LIN {X 0,Y 298.918,Z 266.24,A -85,B 0,C 180,E1 -16378.651,E2 -16378.651} C_VEL
LIN {X 0,Y 298.918,Z 266.244,A -85,B 0,C 180,E1 -16381.346,E2 -16381.346} C_VEL
LIN {X 0,Y 298.79,Z 266.264,A -85,B 0,C 180,E1 -16386.752,E2 -16386.752} C_VEL
LIN {X 0,Y 298.673,Z 266.281,A -85,B 0,C 180,E1 -16389.479,E2 -16389.479} C_VEL
LIN {X 0,Y 298.543,Z 266.299,A -85,B 0,C 180,E1 -16393.614,E2 -16393.614} C_VEL
LIN {X 0,Y 298.54,Z 266.293,A -85,B 0,C 180,E1 -16396.407,E2 -16396.407} C_VEL
LIN {X 0,Y 298.503,Z 266.303,A -85,B 0,C 180,E1 -16399.653,E2 -16399.653} C_VEL
LIN {X 0,Y 298.448,Z 266.307,A -85,B 0,C 180,E1 -16403.596,E2 -16403.596} C_VEL
LIN {X 0,Y 298.48,Z 266.302,A -85,B 0,C 180,E1 -16406.573,E2 -16406.573} C_VEL
LIN {X 0,Y 298.411,Z 266.31,A -85,B 0,C 180,E1 -16409.64,E2 -16409.64} C_VEL
LIN {X 0,Y 298.385,Z 266.316,A -85,B 0,C 180,E1 -16412.799,E2 -16412.799} C_VEL
LIN {X 0,Y 298.456,Z 266.307,A -85,B 0,C 180,E1 -16416.812,E2 -16416.812} C_VEL
LIN {X 0,Y 298.441,Z 266.308,A -85,B 0,C 180,E1 -16421.249,E2 -16421.249} C_VEL
LIN {X 0,Y 298.406,Z 266.315,A -85,B 0,C 180,E1 -16425.046,E2 -16425.046} C_VEL
LIN {X 0,Y 298.378,Z 266.319,A -85,B 0,C 180,E1 -16428.911,E2 -16428.911} C_VEL
LIN {X 0,Y 298.454,Z 266.306,A -85,B 0,C 180,E1 -16433.187,E2 -16433.187} C_VEL
LIN {X 0,Y 298.384,Z 266.315,A -85,B 0,C 180,E1 -16437.199,E2 -16437.199} C_VEL
LIN {X 0,Y 298.414,Z 266.315,A -85,B 0,C 180,E1 -16440.617,E2 -16440.617} C_VEL
LIN {X 0,Y 298.431,Z 266.309,A -85,B 0,C 180,E1 -16443.49,E2 -16443.49} C_VEL
LIN {X 0,Y 298.308,Z 266.328,A -85,B 0,C 180,E1 -16446.749,E2 -16446.749} C_VEL
LIN {X 0,Y 298.289,Z 266.555,A -85,B 0,C 180,E1 -16448.218,E2 -16448.218} C_VEL
LIN {X 0,Y 298.132,Z 269.038,A -85,B 0,C 180,E1 -16450.73,E2 -16450.73} C_VEL
LIN {X 0,Y 297.853,Z 273.686,A -85,B 0,C 180,E1 -16455.325,E2 -16455.325} C_VEL
LIN {X 0,Y 297.53,Z 277.67,A -85,B 0,C 180,E1 -16459.108,E2 -16459.108} C_VEL
LIN {X 0,Y 297.498,Z 279.14,A -85,B 0,C 180,E1 -16460.482,E2 -16460.482} C_VEL
LIN {X 0,Y 301.006,Z 294.207,A -85,B 0,C 180,E1 -16461.43,E2 -16461.43} C_VEL
LIN {X 0,Y 302.952,Z 305.53,A -85,B 0,C 180,E1 -16462.335,E2 -16462.335} C_VEL
LIN {X 0,Y 304.047,Z 314.476,A -85,B 0,C 180,E1 -16463.197,E2 -16463.197} C_VEL
LIN {X 0,Y 303.079,Z 325.319,A -85,B 0,C 180,E1 -16464.344,E2 -16464.344} C_VEL
LIN {X 0,Y 301.711,Z 336.458,A -85,B 0,C 180,E1 -16465.826,E2 -16465.826} C_VEL
LIN {X 0,Y 300.607,Z 345.446,A -85,B 0,C 180,E1 -16467.32,E2 -16467.32} C_VEL
LIN {X 0,Y 299.559,Z 353.696,A -85,B 0,C 180,E1 -16468.992,E2 -16468.992} C_VEL
LIN {X 0,Y 298.399,Z 361.803,A -85,B 0,C 180,E1 -16471.012,E2 -16471.012} C_VEL
LIN {X 0,Y 297.81,Z 367.29,A -85,B 0,C 180,E1 -16472.705,E2 -16472.705} C_VEL
LIN {X 0,Y 297.249,Z 372.668,A -85,B 0,C 180,E1 -16474.747,E2 -16474.747} C_VEL
LIN {X 0,Y 296.913,Z 376.869,A -85,B 0,C 180,E1 -16476.797,E2 -16476.797} C_VEL
LIN {X 0,Y 296.63,Z 379.108,A -85,B 0,C 180,E1 -16478.172,E2 -16478.172} C_VEL
LIN {X 0,Y 296.449,Z 380.852,A -85,B 0,C 180,E1 -16479.552,E2 -16479.552} C_VEL
LIN {X 0,Y 296.349,Z 382.182,A -85,B 0,C 180,E1 -16480.936,E2 -16480.936} C_VEL
LIN {X 0,Y 296.375,Z 383.581,A -85,B 0,C 180,E1 -16483.541,E2 -16483.541} C_VEL
LIN {X 0,Y 296.381,Z 383.689,A -85,B 0,C 180,E1 -16485.119,E2 -16485.119} C_VEL
LIN {X 0,Y 296.494,Z 383.364,A -85,B 0,C 180,E1 -16486.525,E2 -16486.525} C_VEL
LIN {X 0,Y 296.901,Z 381.967,A -85,B 0,C 180,E1 -16488.772,E2 -16488.772} C_VEL
LIN {X 0,Y 297.663,Z 378.824,A -85,B 0,C 180,E1 -16491.466,E2 -16491.466} C_VEL
LIN {X 0,Y 298.539,Z 375.125,A -85,B 0,C 180,E1 -16493.59,E2 -16493.59} C_VEL
LIN {X 0,Y 299.663,Z 370.217,A -85,B 0,C 180,E1 -16495.713,E2 -16495.713} C_VEL
LIN {X 0,Y 301.161,Z 363.948,A -85,B 0,C 180,E1 -16497.821,E2 -16497.821} C_VEL
LIN {X 0,Y 302.967,Z 356.064,A -85,B 0,C 180,E1 -16499.916,E2 -16499.916} C_VEL
LIN {X 0,Y 304.904,Z 347.289,A -85,B 0,C 180,E1 -16501.752,E2 -16501.752} C_VEL
LIN {X 0,Y 306.788,Z 337.818,A -85,B 0,C 180,E1 -16503.352,E2 -16503.352} C_VEL
LIN {X 0,Y 308.587,Z 327.879,A -85,B 0,C 180,E1 -16504.705,E2 -16504.705} C_VEL
LIN {X 0,Y 309.544,Z 321.191,A -85,B 0,C 180,E1 -16505.475,E2 -16505.475} C_VEL
LIN {X 0,Y 307.576,Z 309.692,A -85,B 0,C 180,E1 -16506.898,E2 -16506.898} C_VEL
LIN {X 0,Y 304.312,Z 297.366,A -85,B 0,C 180,E1 -16508.262,E2 -16508.262} C_VEL
LIN {X 0,Y 300.102,Z 285.47,A -85,B 0,C 180,E1 -16509.441,E2 -16509.441} C_VEL
LIN {X 0,Y 298.087,Z 279.79,A -85,B 0,C 180,E1 -16509.934,E2 -16509.934} C_VEL
LIN {X 0,Y 298.415,Z 276.805,A -85,B 0,C 180,E1 -16513.11,E2 -16513.11} C_VEL
LIN {X 0,Y 298.864,Z 273.306,A -85,B 0,C 180,E1 -16517.006,E2 -16517.006} C_VEL
LIN {X 0,Y 298.92,Z 271.733,A -85,B 0,C 180,E1 -16518.831,E2 -16518.831} C_VEL
LIN {X 0,Y 298.715,Z 268.955,A -85,B 0,C 180,E1 -16522.289,E2 -16522.289} C_VEL
LIN {X 0,Y 298.42,Z 266.485,A -85,B 0,C 180,E1 -16525.585,E2 -16525.585} C_VEL
LIN {X 0,Y 298.384,Z 266.322,A -85,B 0,C 180,E1 -16528.792,E2 -16528.792} C_VEL
LIN {X 0,Y 298.453,Z 266.311,A -85,B 0,C 180,E1 -16531.905,E2 -16531.905} C_VEL
LIN {X 0,Y 298.478,Z 266.304,A -85,B 0,C 180,E1 -16534.925,E2 -16534.925} C_VEL
LIN {X 0,Y 298.46,Z 266.305,A -85,B 0,C 180,E1 -16539.318,E2 -16539.318} C_VEL
LIN {X 0,Y 298.53,Z 266.295,A -85,B 0,C 180,E1 -16542.181,E2 -16542.181} C_VEL
LIN {X 0,Y 298.537,Z 266.294,A -85,B 0,C 180,E1 -16546.12,E2 -16546.12} C_VEL
LIN {X 0,Y 298.627,Z 266.288,A -85,B 0,C 180,E1 -16550.52,E2 -16550.52} C_VEL
LIN {X 0,Y 298.73,Z 266.273,A -85,B 0,C 180,E1 -16551.968,E2 -16551.968} C_VEL
LIN {X 0,Y 298.053,Z 266.359,A -85,B 0,C 180,E1 -16553.092,E2 -16553.092} C_VEL
LIN {X 0,Y 295.209,Z 266.713,A -85,B 0,C 180,E1 -16554.923,E2 -16554.923} C_VEL
LIN {X 0,Y 292.837,Z 267.009,A -85,B 0,C 180,E1 -16556.409,E2 -16556.409} C_VEL
LIN {X 0,Y 291.867,Z 267.129,A -85,B 0,C 180,E1 -16557.56,E2 -16557.56} C_VEL
LIN {X 0,Y 291.812,Z 267.134,A -85,B 0,C 180,E1 -16557.949,E2 -16557.949} C_VEL
LIN {X 0,Y 291.944,Z 267.118,A -85,B 0,C 180,E1 -16560.002,E2 -16560.002} C_VEL
LIN {X 0,Y 291.783,Z 267.14,A -85,B 0,C 180,E1 -16562.763,E2 -16562.763} C_VEL
LIN {X 0,Y 291.739,Z 267.146,A -85,B 0,C 180,E1 -16566.92,E2 -16566.92} C_VEL
LIN {X 0,Y 291.624,Z 267.159,A -85,B 0,C 180,E1 -16569.714,E2 -16569.714} C_VEL
LIN {X 0,Y 291.517,Z 267.174,A -85,B 0,C 180,E1 -16573.952,E2 -16573.952} C_VEL
LIN {X 0,Y 291.483,Z 267.181,A -85,B 0,C 180,E1 -16576.82,E2 -16576.82} C_VEL
LIN {X 0,Y 291.448,Z 267.187,A -85,B 0,C 180,E1 -16579.877,E2 -16579.877} C_VEL
LIN {X 0,Y 291.369,Z 267.197,A -85,B 0,C 180,E1 -16584.21,E2 -16584.21} C_VEL
LIN {X 0,Y 291.393,Z 267.195,A -85,B 0,C 180,E1 -16587.276,E2 -16587.276} C_VEL
LIN {X 0,Y 291.319,Z 267.202,A -85,B 0,C 180,E1 -16590.44,E2 -16590.44} C_VEL
LIN {X 0,Y 291.342,Z 267.196,A -85,B 0,C 180,E1 -16593.7,E2 -16593.7} C_VEL
LIN {X 0,Y 291.375,Z 267.191,A -85,B 0,C 180,E1 -16597.255,E2 -16597.255} C_VEL
LIN {X 0,Y 291.379,Z 267.265,A -85,B 0,C 180,E1 -16598.411,E2 -16598.411} C_VEL
LIN {X 0,Y 291.89,Z 270.67,A -85,B 0,C 180,E1 -16602.392,E2 -16602.392} C_VEL
LIN {X 0,Y 292.517,Z 274.169,A -85,B 0,C 180,E1 -16606.121,E2 -16606.121} C_VEL
LIN {X 0,Y 293.083,Z 277.742,A -85,B 0,C 180,E1 -16609.652,E2 -16609.652} C_VEL
LIN {X 0,Y 293.435,Z 281.675,A -85,B 0,C 180,E1 -16613.219,E2 -16613.219} C_VEL
LIN {X 0,Y 293.336,Z 283.651,A -85,B 0,C 180,E1 -16614.901,E2 -16614.901} C_VEL
LIN {X 0,Y 292.655,Z 287.637,A -85,B 0,C 180,E1 -16618.109,E2 -16618.109} C_VEL
LIN {X 0,Y 291.73,Z 293.108,A -85,B 0,C 180,E1 -16622.337,E2 -16622.337} C_VEL
LIN {X 0,Y 292.705,Z 296.464,A -85,B 0,C 180,E1 -16622.601,E2 -16622.601} C_VEL
LIN {X 0,Y 296.744,Z 309.875,A -85,B 0,C 180,E1 -16623.81,E2 -16623.81} C_VEL
LIN {X 0,Y 299.461,Z 322.339,A -85,B 0,C 180,E1 -16625.088,E2 -16625.088} C_VEL
LIN {X 0,Y 301.014,Z 333.959,A -85,B 0,C 180,E1 -16626.455,E2 -16626.455} C_VEL
LIN {X 0,Y 301.385,Z 342.41,A -85,B 0,C 180,E1 -16627.552,E2 -16627.552} C_VEL
LIN {X 0,Y 299.351,Z 353.181,A -85,B 0,C 180,E1 -16629.021,E2 -16629.021} C_VEL
LIN {X 0,Y 297.151,Z 362.889,A -85,B 0,C 180,E1 -16630.664,E2 -16630.664} C_VEL
LIN {X 0,Y 295.31,Z 371.442,A -85,B 0,C 180,E1 -16632.477,E2 -16632.477} C_VEL
LIN {X 0,Y 293.712,Z 378.715,A -85,B 0,C 180,E1 -16634.384,E2 -16634.384} C_VEL
LIN {X 0,Y 292.344,Z 384.053,A -85,B 0,C 180,E1 -16636.09,E2 -16636.09} C_VEL
LIN {X 0,Y 291.181,Z 389.297,A -85,B 0,C 180,E1 -16638.162,E2 -16638.162} C_VEL
LIN {X 0,Y 290.347,Z 393.396,A -85,B 0,C 180,E1 -16640.245,E2 -16640.245} C_VEL
LIN {X 0,Y 289.935,Z 395.563,A -85,B 0,C 180,E1 -16641.638,E2 -16641.638} C_VEL
LIN {X 0,Y 289.482,Z 398.581,A -85,B 0,C 180,E1 -16644.427,E2 -16644.427} C_VEL
LIN {X 0,Y 289.406,Z 399.505,A -85,B 0,C 180,E1 -16645.822,E2 -16645.822} C_VEL
LIN {X 0,Y 289.433,Z 400.027,A -85,B 0,C 180,E1 -16647.217,E2 -16647.217} C_VEL
LIN {X 0,Y 289.409,Z 400.124,A -85,B 0,C 180,E1 -16648.609,E2 -16648.609} C_VEL
LIN {X 0,Y 289.439,Z 399.839,A -85,B 0,C 180,E1 -16650,E2 -16650} C_VEL
LIN {X 0,Y 289.423,Z 399.164,A -85,B 0,C 180,E1 -16651.391,E2 -16651.391} C_VEL
LIN {X 0,Y 289.47,Z 398.086,A -85,B 0,C 180,E1 -16652.783,E2 -16652.783} C_VEL
LIN {X 0,Y 289.445,Z 396.547,A -85,B 0,C 180,E1 -16654.177,E2 -16654.177} C_VEL
LIN {X 0,Y 289.564,Z 393.444,A -85,B 0,C 180,E1 -16656.27,E2 -16656.27} C_VEL
LIN {X 0,Y 289.839,Z 389.262,A -85,B 0,C 180,E1 -16658.365,E2 -16658.365} C_VEL
LIN {X 0,Y 290.461,Z 382.866,A -85,B 0,C 180,E1 -16660.808,E2 -16660.808} C_VEL
LIN {X 0,Y 291.276,Z 375.883,A -85,B 0,C 180,E1 -16662.896,E2 -16662.896} C_VEL
LIN {X 0,Y 292.21,Z 368.739,A -85,B 0,C 180,E1 -16664.627,E2 -16664.627} C_VEL
LIN {X 0,Y 293.307,Z 359.865,A -85,B 0,C 180,E1 -16666.39,E2 -16666.39} C_VEL
LIN {X 0,Y 294.579,Z 349.371,A -85,B 0,C 180,E1 -16668.068,E2 -16668.068} C_VEL
LIN {X 0,Y 295.97,Z 338.769,A -85,B 0,C 180,E1 -16669.416,E2 -16669.416} C_VEL
LIN {X 0,Y 295.933,Z 333.974,A -85,B 0,C 180,E1 -16669.961,E2 -16669.961} C_VEL
LIN {X 0,Y 294.798,Z 321.713,A -85,B 0,C 180,E1 -16671.185,E2 -16671.185} C_VEL
LIN {X 0,Y 293.106,Z 308.712,A -85,B 0,C 180,E1 -16672.196,E2 -16672.196} C_VEL
LIN {X 0,Y 290.789,Z 295.542,A -85,B 0,C 180,E1 -16672.971,E2 -16672.971} C_VEL
LIN {X 0,Y 290.508,Z 293.683,A -85,B 0,C 180,E1 -16673.097,E2 -16673.097} C_VEL
LIN {X 0,Y 291.1,Z 287.723,A -85,B 0,C 180,E1 -16677.304,E2 -16677.304} C_VEL
LIN {X 0,Y 291.952,Z 281.246,A -85,B 0,C 180,E1 -16681.977,E2 -16681.977} C_VEL
LIN {X 0,Y 292.563,Z 276.873,A -85,B 0,C 180,E1 -16685.237,E2 -16685.237} C_VEL
LIN {X 0,Y 292.569,Z 273.875,A -85,B 0,C 180,E1 -16687.558,E2 -16687.558} C_VEL
LIN {X 0,Y 291.704,Z 268.923,A -85,B 0,C 180,E1 -16691.677,E2 -16691.677} C_VEL
LIN {X 0,Y 291.356,Z 267.194,A -85,B 0,C 180,E1 -16693.335,E2 -16693.335} C_VEL
LIN {X 0,Y 291.283,Z 267.203,A -85,B 0,C 180,E1 -16697.499,E2 -16697.499} C_VEL
LIN {X 0,Y 291.331,Z 267.197,A -85,B 0,C 180,E1 -16701.153,E2 -16701.153} C_VEL
LIN {X 0,Y 291.353,Z 267.195,A -85,B 0,C 180,E1 -16704.623,E2 -16704.623} C_VEL
LIN {X 0,Y 291.364,Z 267.189,A -85,B 0,C 180,E1 -16707.948,E2 -16707.948} C_VEL
LIN {X 0,Y 291.341,Z 267.192,A -85,B 0,C 180,E1 -16711.152,E2 -16711.152} C_VEL
LIN {X 0,Y 291.356,Z 267.193,A -85,B 0,C 180,E1 -16714.265,E2 -16714.265} C_VEL
LIN {X 0,Y 291.363,Z 267.189,A -85,B 0,C 180,E1 -16717.296,E2 -16717.296} C_VEL
LIN {X 0,Y 291.455,Z 267.182,A -85,B 0,C 180,E1 -16720.268,E2 -16720.268} C_VEL
LIN {X 0,Y 291.537,Z 267.17,A -85,B 0,C 180,E1 -16724.633,E2 -16724.633} C_VEL
LIN {X 0,Y 291.53,Z 267.167,A -85,B 0,C 180,E1 -16728.879,E2 -16728.879} C_VEL
LIN {X 0,Y 291.683,Z 267.151,A -85,B 0,C 180,E1 -16731.686,E2 -16731.686} C_VEL
LIN {X 0,Y 291.621,Z 267.157,A -85,B 0,C 180,E1 -16734.467,E2 -16734.467} C_VEL
LIN {X 0,Y 291.884,Z 267.115,A -85,B 0,C 180,E1 -16738.619,E2 -16738.619} C_VEL
LIN {X 0,Y 291.885,Z 267.119,A -85,B 0,C 180,E1 -16741.378,E2 -16741.378} C_VEL
LIN {X 0,Y 291.739,Z 267.142,A -85,B 0,C 180,E1 -16746.916,E2 -16746.916} C_VEL
LIN {X 0,Y 291.622,Z 267.159,A -85,B 0,C 180,E1 -16749.71,E2 -16749.71} C_VEL
LIN {X 0,Y 291.513,Z 267.172,A -85,B 0,C 180,E1 -16753.949,E2 -16753.949} C_VEL
LIN {X 0,Y 291.478,Z 267.173,A -85,B 0,C 180,E1 -16756.816,E2 -16756.816} C_VEL
LIN {X 0,Y 291.442,Z 267.181,A -85,B 0,C 180,E1 -16759.873,E2 -16759.873} C_VEL
LIN {X 0,Y 291.391,Z 267.183,A -85,B 0,C 180,E1 -16764.204,E2 -16764.204} C_VEL
LIN {X 0,Y 291.413,Z 267.187,A -85,B 0,C 180,E1 -16767.27,E2 -16767.27} C_VEL
LIN {X 0,Y 291.328,Z 267.191,A -85,B 0,C 180,E1 -16770.436,E2 -16770.436} C_VEL
LIN {X 0,Y 291.335,Z 267.193,A -85,B 0,C 180,E1 -16773.697,E2 -16773.697} C_VEL
LIN {X 0,Y 291.389,Z 267.188,A -85,B 0,C 180,E1 -16777.259,E2 -16777.259} C_VEL
LIN {X 0,Y 291.39,Z 267.188,A -85,B 0,C 180,E1 -16780.63,E2 -16780.63} C_VEL
LIN {X 0,Y 291.342,Z 267.192,A -85,B 0,C 180,E1 -16784.389,E2 -16784.389} C_VEL
LIN {X 0,Y 291.321,Z 267.194,A -85,B 0,C 180,E1 -16788.402,E2 -16788.402} C_VEL
LIN {X 0,Y 291.343,Z 267.192,A -85,B 0,C 180,E1 -16791.158,E2 -16791.158} C_VEL
LIN {X 0,Y 291.375,Z 267.193,A -85,B 0,C 180,E1 -16794.629,E2 -16794.629} C_VEL
LIN {X 0,Y 291.359,Z 267.191,A -85,B 0,C 180,E1 -16797.95,E2 -16797.95} C_VEL
LIN {X 0,Y 291.358,Z 267.19,A -85,B 0,C 180,E1 -16801.156,E2 -16801.156} C_VEL
LIN {X 0,Y 291.354,Z 267.194,A -85,B 0,C 180,E1 -16804.267,E2 -16804.267} C_VEL
LIN {X 0,Y 291.293,Z 267.305,A -85,B 0,C 180,E1 -16808.04,E2 -16808.04} C_VEL
LIN {X 0,Y 290.956,Z 270.87,A -85,B 0,C 180,E1 -16811.699,E2 -16811.699} C_VEL
LIN {X 0,Y 290.72,Z 275.198,A -85,B 0,C 180,E1 -16816.011,E2 -16816.011} C_VEL
LIN {X 0,Y 290.437,Z 279.352,A -85,B 0,C 180,E1 -16820.028,E2 -16820.028} C_VEL
LIN {X 0,Y 293.921,Z 293.917,A -85,B 0,C 180,E1 -16820.969,E2 -16820.969} C_VEL
LIN {X 0,Y 296.064,Z 306.265,A -85,B 0,C 180,E1 -16821.983,E2 -16821.983} C_VEL
LIN {X 0,Y 297.199,Z 316.77,A -85,B 0,C 180,E1 -16823.039,E2 -16823.039} C_VEL
LIN {X 0,Y 295.841,Z 328.512,A -85,B 0,C 180,E1 -16824.376,E2 -16824.376} C_VEL
LIN {X 0,Y 294.493,Z 339.037,A -85,B 0,C 180,E1 -16825.894,E2 -16825.894} C_VEL
LIN {X 0,Y 293.248,Z 348.521,A -85,B 0,C 180,E1 -16827.596,E2 -16827.596} C_VEL
LIN {X 0,Y 292.035,Z 357.643,A -85,B 0,C 180,E1 -16829.655,E2 -16829.655} C_VEL
LIN {X 0,Y 291.013,Z 365.006,A -85,B 0,C 180,E1 -16831.73,E2 -16831.73} C_VEL
LIN {X 0,Y 290.457,Z 369.991,A -85,B 0,C 180,E1 -16833.468,E2 -16833.468} C_VEL
LIN {X 0,Y 290.011,Z 374.834,A -85,B 0,C 180,E1 -16835.562,E2 -16835.562} C_VEL
LIN {X 0,Y 289.641,Z 378.568,A -85,B 0,C 180,E1 -16837.669,E2 -16837.669} C_VEL
LIN {X 0,Y 289.332,Z 381.283,A -85,B 0,C 180,E1 -16839.789,E2 -16839.789} C_VEL
LIN {X 0,Y 289.265,Z 382.561,A -85,B 0,C 180,E1 -16841.207,E2 -16841.207} C_VEL
LIN {X 0,Y 289.284,Z 383.782,A -85,B 0,C 180,E1 -16843.654,E2 -16843.654} C_VEL
LIN {X 0,Y 289.308,Z 383.868,A -85,B 0,C 180,E1 -16845.498,E2 -16845.498} C_VEL
LIN {X 0,Y 289.457,Z 383.493,A -85,B 0,C 180,E1 -16846.939,E2 -16846.939} C_VEL
LIN {X 0,Y 289.857,Z 382.191,A -85,B 0,C 180,E1 -16848.991,E2 -16848.991} C_VEL
LIN {X 0,Y 290.756,Z 378.689,A -85,B 0,C 180,E1 -16852.003,E2 -16852.003} C_VEL
LIN {X 0,Y 291.745,Z 374.873,A -85,B 0,C 180,E1 -16854.174,E2 -16854.174} C_VEL
LIN {X 0,Y 292.983,Z 369.841,A -85,B 0,C 180,E1 -16856.344,E2 -16856.344} C_VEL
LIN {X 0,Y 294.605,Z 363.436,A -85,B 0,C 180,E1 -16858.496,E2 -16858.496} C_VEL
LIN {X 0,Y 296.177,Z 356.815,A -85,B 0,C 180,E1 -16860.28,E2 -16860.28} C_VEL
LIN {X 0,Y 298.24,Z 347.959,A -85,B 0,C 180,E1 -16862.199,E2 -16862.199} C_VEL
LIN {X 0,Y 300.393,Z 337.762,A -85,B 0,C 180,E1 -16863.957,E2 -16863.957} C_VEL
LIN {X 0,Y 302.262,Z 327.768,A -85,B 0,C 180,E1 -16865.335,E2 -16865.335} C_VEL
LIN {X 0,Y 302.962,Z 323.772,A -85,B 0,C 180,E1 -16865.802,E2 -16865.802} C_VEL
LIN {X 0,Y 302.229,Z 317.404,A -85,B 0,C 180,E1 -16866.658,E2 -16866.658} C_VEL
LIN {X 0,Y 300.306,Z 307.817,A -85,B 0,C 180,E1 -16867.854,E2 -16867.854} C_VEL
LIN {X 0,Y 297.266,Z 296.818,A -85,B 0,C 180,E1 -16869.098,E2 -16869.098} C_VEL
LIN {X 0,Y 292.499,Z 283.66,A -85,B 0,C 180,E1 -16870.43,E2 -16870.43} C_VEL
LIN {X 0,Y 291.299,Z 280.869,A -85,B 0,C 180,E1 -16870.707,E2 -16870.707} C_VEL
LIN {X 0,Y 291.157,Z 279.995,A -85,B 0,C 180,E1 -16870.796,E2 -16870.796} C_VEL
LIN {X 0,Y 291.511,Z 276.756,A -85,B 0,C 180,E1 -16874.358,E2 -16874.358} C_VEL
LIN {X 0,Y 291.862,Z 273.931,A -85,B 0,C 180,E1 -16877.608,E2 -16877.608} C_VEL
LIN {X 0,Y 291.817,Z 271.01,A -85,B 0,C 180,E1 -16881.234,E2 -16881.234} C_VEL
LIN {X 0,Y 291.497,Z 268.156,A -85,B 0,C 180,E1 -16885.057,E2 -16885.057} C_VEL
LIN {X 0,Y 291.346,Z 267.287,A -85,B 0,C 180,E1 -16886.304,E2 -16886.304} C_VEL
LIN {X 0,Y 291.377,Z 267.193,A -85,B 0,C 180,E1 -16890.261,E2 -16890.261} C_VEL
LIN {X 0,Y 291.409,Z 267.187,A -85,B 0,C 180,E1 -16894.273,E2 -16894.273} C_VEL
LIN {X 0,Y 291.39,Z 267.185,A -85,B 0,C 180,E1 -16897.302,E2 -16897.302} C_VEL
LIN {X 0,Y 291.495,Z 267.174,A -85,B 0,C 180,E1 -16900.275,E2 -16900.275} C_VEL
LIN {X 0,Y 291.532,Z 267.17,A -85,B 0,C 180,E1 -16904.636,E2 -16904.636} C_VEL
LIN {X 0,Y 291.527,Z 267.172,A -85,B 0,C 180,E1 -16908.882,E2 -16908.882} C_VEL
LIN {X 0,Y 291.675,Z 267.151,A -85,B 0,C 180,E1 -16911.967,E2 -16911.967} C_VEL
LIN {X 0,Y 291.619,Z 267.161,A -85,B 0,C 180,E1 -16914.47,E2 -16914.47} C_VEL
LIN {X 0,Y 291.812,Z 267.134,A -85,B 0,C 180,E1 -16917.949,E2 -16917.949} C_VEL
LIN {X 0,Y 291.205,Z 267.212,A -85,B 0,C 180,E1 -16919.102,E2 -16919.102} C_VEL
LIN {X 0,Y 288.33,Z 267.57,A -85,B 0,C 180,E1 -16920.977,E2 -16920.977} C_VEL
LIN {X 0,Y 285.802,Z 267.885,A -85,B 0,C 180,E1 -16922.499,E2 -16922.499} C_VEL
LIN {X 0,Y 284.649,Z 268.028,A -85,B 0,C 180,E1 -16923.679,E2 -16923.679} C_VEL
LIN {X 0,Y 284.521,Z 268.043,A -85,B 0,C 180,E1 -16924.081,E2 -16924.081} C_VEL
LIN {X 0,Y 284.692,Z 268.023,A -85,B 0,C 180,E1 -16927.092,E2 -16927.092} C_VEL
LIN {X 0,Y 284.561,Z 268.039,A -85,B 0,C 180,E1 -16929.957,E2 -16929.957} C_VEL
LIN {X 0,Y 284.473,Z 268.054,A -85,B 0,C 180,E1 -16934.305,E2 -16934.305} C_VEL
LIN {X 0,Y 284.421,Z 268.06,A -85,B 0,C 180,E1 -16937.25,E2 -16937.25} C_VEL
LIN {X 0,Y 284.376,Z 268.068,A -85,B 0,C 180,E1 -16940.244,E2 -16940.244} C_VEL
LIN {X 0,Y 284.319,Z 268.076,A -85,B 0,C 180,E1 -16944.85,E2 -16944.85} C_VEL
LIN {X 0,Y 284.304,Z 268.077,A -85,B 0,C 180,E1 -16948.015,E2 -16948.015} C_VEL
LIN {X 0,Y 284.284,Z 268.078,A -85,B 0,C 180,E1 -16951.277,E2 -16951.277} C_VEL
LIN {X 0,Y 284.34,Z 268.067,A -85,B 0,C 180,E1 -16955.35,E2 -16955.35} C_VEL
LIN {X 0,Y 284.359,Z 268.264,A -85,B 0,C 180,E1 -16957.733,E2 -16957.733} C_VEL
LIN {X 0,Y 284.689,Z 270.141,A -85,B 0,C 180,E1 -16960.069,E2 -16960.069} C_VEL
LIN {X 0,Y 285.256,Z 273.914,A -85,B 0,C 180,E1 -16964.4,E2 -16964.4} C_VEL
LIN {X 0,Y 285.922,Z 277.77,A -85,B 0,C 180,E1 -16968.421,E2 -16968.421} C_VEL
LIN {X 0,Y 286.427,Z 281.698,A -85,B 0,C 180,E1 -16972.164,E2 -16972.164} C_VEL
LIN {X 0,Y 286.373,Z 283.86,A -85,B 0,C 180,E1 -16974.085,E2 -16974.085} C_VEL
LIN {X 0,Y 285.837,Z 287.621,A -85,B 0,C 180,E1 -16977.254,E2 -16977.254} C_VEL
LIN {X 0,Y 284.839,Z 292.896,A -85,B 0,C 180,E1 -16981.465,E2 -16981.465} C_VEL
LIN {X 0,Y 285.781,Z 296.152,A -85,B 0,C 180,E1 -16981.723,E2 -16981.723} C_VEL
LIN {X 0,Y 289.823,Z 309.168,A -85,B 0,C 180,E1 -16982.962,E2 -16982.962} C_VEL
LIN {X 0,Y 292.471,Z 320.562,A -85,B 0,C 180,E1 -16984.174,E2 -16984.174} C_VEL
LIN {X 0,Y 294.185,Z 332.406,A -85,B 0,C 180,E1 -16985.581,E2 -16985.581} C_VEL
LIN {X 0,Y 294.795,Z 341.735,A -85,B 0,C 180,E1 -16986.837,E2 -16986.837} C_VEL
LIN {X 0,Y 294.451,Z 345.58,A -85,B 0,C 180,E1 -16987.365,E2 -16987.365} C_VEL
LIN {X 0,Y 292.241,Z 355.763,A -85,B 0,C 180,E1 -16988.856,E2 -16988.856} C_VEL
LIN {X 0,Y 290.058,Z 364.936,A -85,B 0,C 180,E1 -16990.54,E2 -16990.54} C_VEL
LIN {X 0,Y 288.311,Z 372.947,A -85,B 0,C 180,E1 -16992.378,E2 -16992.378} C_VEL
LIN {X 0,Y 286.582,Z 379.973,A -85,B 0,C 180,E1 -16994.351,E2 -16994.351} C_VEL
LIN {X 0,Y 284.968,Z 385.995,A -85,B 0,C 180,E1 -16996.45,E2 -16996.45} C_VEL
LIN {X 0,Y 283.873,Z 390.783,A -85,B 0,C 180,E1 -16998.577,E2 -16998.577} C_VEL
LIN {X 0,Y 283.102,Z 394.477,A -85,B 0,C 180,E1 -17000.714,E2 -17000.714} C_VEL
LIN {X 0,Y 282.588,Z 397.178,A -85,B 0,C 180,E1 -17002.857,E2 -17002.857} C_VEL
LIN {X 0,Y 282.401,Z 398.677,A -85,B 0,C 180,E1 -17004.553,E2 -17004.553} C_VEL
LIN {X 0,Y 282.339,Z 399.838,A -85,B 0,C 180,E1 -17007.147,E2 -17007.147} C_VEL
LIN {X 0,Y 282.333,Z 399.912,A -85,B 0,C 180,E1 -17008.574,E2 -17008.574} C_VEL
LIN {X 0,Y 282.358,Z 399.602,A -85,B 0,C 180,E1 -17010,E2 -17010} C_VEL
LIN {X 0,Y 282.346,Z 398.904,A -85,B 0,C 180,E1 -17011.426,E2 -17011.426} C_VEL
LIN {X 0,Y 282.375,Z 397.778,A -85,B 0,C 180,E1 -17012.853,E2 -17012.853} C_VEL
LIN {X 0,Y 282.413,Z 394.583,A -85,B 0,C 180,E1 -17015.474,E2 -17015.474} C_VEL
LIN {X 0,Y 282.673,Z 390.358,A -85,B 0,C 180,E1 -17017.859,E2 -17017.859} C_VEL
LIN {X 0,Y 283.127,Z 385.342,A -85,B 0,C 180,E1 -17020.006,E2 -17020.006} C_VEL
LIN {X 0,Y 283.796,Z 379.02,A -85,B 0,C 180,E1 -17022.151,E2 -17022.151} C_VEL
LIN {X 0,Y 284.94,Z 371.097,A -85,B 0,C 180,E1 -17024.279,E2 -17024.279} C_VEL
LIN {X 0,Y 286.143,Z 361.996,A -85,B 0,C 180,E1 -17026.242,E2 -17026.242} C_VEL
LIN {X 0,Y 287.369,Z 351.995,A -85,B 0,C 180,E1 -17027.984,E2 -17027.984} C_VEL
LIN {X 0,Y 288.671,Z 342.007,A -85,B 0,C 180,E1 -17029.372,E2 -17029.372} C_VEL
LIN {X 0,Y 289.22,Z 337.68,A -85,B 0,C 180,E1 -17029.888,E2 -17029.888} C_VEL
LIN {X 0,Y 288.286,Z 325.951,A -85,B 0,C 180,E1 -17031.182,E2 -17031.182} C_VEL
LIN {X 0,Y 286.91,Z 313.75,A -85,B 0,C 180,E1 -17032.258,E2 -17032.258} C_VEL
LIN {X 0,Y 284.839,Z 300.778,A -85,B 0,C 180,E1 -17033.149,E2 -17033.149} C_VEL
LIN {X 0,Y 283.475,Z 293.526,A -85,B 0,C 180,E1 -17033.544,E2 -17033.544} C_VEL
LIN {X 0,Y 284.116,Z 287.357,A -85,B 0,C 180,E1 -17038.033,E2 -17038.033} C_VEL
LIN {X 0,Y 284.915,Z 281.979,A -85,B 0,C 180,E1 -17042.028,E2 -17042.028} C_VEL
LIN {X 0,Y 285.555,Z 277.196,A -85,B 0,C 180,E1 -17045.688,E2 -17045.688} C_VEL
LIN {X 0,Y 285.449,Z 274.292,A -85,B 0,C 180,E1 -17048.011,E2 -17048.011} C_VEL
LIN {X 0,Y 284.615,Z 269.424,A -85,B 0,C 180,E1 -17052.199,E2 -17052.199} C_VEL
LIN {X 0,Y 284.317,Z 268.071,A -85,B 0,C 180,E1 -17053.487,E2 -17053.487} C_VEL
LIN {X 0,Y 284.233,Z 268.081,A -85,B 0,C 180,E1 -17058.116,E2 -17058.116} C_VEL
LIN {X 0,Y 284.292,Z 268.072,A -85,B 0,C 180,E1 -17061.826,E2 -17061.826} C_VEL
LIN {X 0,Y 284.305,Z 268.069,A -85,B 0,C 180,E1 -17065.349,E2 -17065.349} C_VEL
LIN {X 0,Y 284.283,Z 268.074,A -85,B 0,C 180,E1 -17068.723,E2 -17068.723} C_VEL
LIN {X 0,Y 284.281,Z 268.072,A -85,B 0,C 180,E1 -17071.982,E2 -17071.982} C_VEL
LIN {X 0,Y 284.318,Z 268.068,A -85,B 0,C 180,E1 -17076.145,E2 -17076.145} C_VEL
LIN {X 0,Y 284.385,Z 268.06,A -85,B 0,C 180,E1 -17079.896,E2 -17079.896} C_VEL
LIN {X 0,Y 284.475,Z 268.051,A -85,B 0,C 180,E1 -17084.468,E2 -17084.468} C_VEL
LIN {X 0,Y 284.482,Z 268.046,A -85,B 0,C 180,E1 -17088.6,E2 -17088.6} C_VEL
LIN {X 0,Y 284.634,Z 268.028,A -85,B 0,C 180,E1 -17091.479,E2 -17091.479} C_VEL
LIN {X 0,Y 284.591,Z 268.034,A -85,B 0,C 180,E1 -17094.329,E2 -17094.329} C_VEL
LIN {X 0,Y 284.85,Z 267.99,A -85,B 0,C 180,E1 -17098.585,E2 -17098.585} C_VEL
LIN {X 0,Y 284.85,Z 267.995,A -85,B 0,C 180,E1 -17101.412,E2 -17101.412} C_VEL
LIN {X 0,Y 284.691,Z 268.021,A -85,B 0,C 180,E1 -17107.088,E2 -17107.088} C_VEL
LIN {X 0,Y 284.559,Z 268.037,A -85,B 0,C 180,E1 -17109.954,E2 -17109.954} C_VEL
LIN {X 0,Y 284.47,Z 268.048,A -85,B 0,C 180,E1 -17114.301,E2 -17114.301} C_VEL
LIN {X 0,Y 284.417,Z 268.055,A -85,B 0,C 180,E1 -17117.247,E2 -17117.247} C_VEL
LIN {X 0,Y 284.37,Z 268.06,A -85,B 0,C 180,E1 -17120.241,E2 -17120.241} C_VEL
LIN {X 0,Y 284.36,Z 268.06,A -85,B 0,C 180,E1 -17123.874,E2 -17123.874} C_VEL
LIN {X 0,Y 284.388,Z 268.062,A -85,B 0,C 180,E1 -17127.172,E2 -17127.172} C_VEL
LIN {X 0,Y 284.286,Z 268.073,A -85,B 0,C 180,E1 -17131.273,E2 -17131.273} C_VEL
LIN {X 0,Y 284.352,Z 268.063,A -85,B 0,C 180,E1 -17135.353,E2 -17135.353} C_VEL
LIN {X 0,Y 284.321,Z 268.065,A -85,B 0,C 180,E1 -17138.165,E2 -17138.165} C_VEL
LIN {X 0,Y 284.33,Z 268.063,A -85,B 0,C 180,E1 -17142.139,E2 -17142.139} C_VEL
LIN {X 0,Y 284.286,Z 268.071,A -85,B 0,C 180,E1 -17146.196,E2 -17146.196} C_VEL
LIN {X 0,Y 284.296,Z 268.07,A -85,B 0,C 180,E1 -17150.023,E2 -17150.023} C_VEL
LIN {X 0,Y 284.337,Z 268.064,A -85,B 0,C 180,E1 -17153.616,E2 -17153.616} C_VEL
LIN {X 0,Y 284.297,Z 268.07,A -85,B 0,C 180,E1 -17157.189,E2 -17157.189} C_VEL
LIN {X 0,Y 284.343,Z 268.068,A -85,B 0,C 180,E1 -17160.375,E2 -17160.375} C_VEL
LIN {X 0,Y 284.335,Z 268.065,A -85,B 0,C 180,E1 -17163.583,E2 -17163.583} C_VEL
LIN {X 0,Y 284.265,Z 268.232,A -85,B 0,C 180,E1 -17168.042,E2 -17168.042} C_VEL
LIN {X 0,Y 283.953,Z 271.263,A -85,B 0,C 180,E1 -17171.231,E2 -17171.231} C_VEL
LIN {X 0,Y 283.682,Z 275.615,A -85,B 0,C 180,E1 -17175.656,E2 -17175.656} C_VEL
LIN {X 0,Y 283.383,Z 279.567,A -85,B 0,C 180,E1 -17179.554,E2 -17179.554} C_VEL
LIN {X 0,Y 286.792,Z 293.525,A -85,B 0,C 180,E1 -17180.475,E2 -17180.475} C_VEL
LIN {X 0,Y 289.007,Z 305.951,A -85,B 0,C 180,E1 -17181.519,E2 -17181.519} C_VEL
LIN {X 0,Y 290.253,Z 315.704,A -85,B 0,C 180,E1 -17182.522,E2 -17182.522} C_VEL
LIN {X 0,Y 289.816,Z 322.077,A -85,B 0,C 180,E1 -17183.211,E2 -17183.211} C_VEL
LIN {X 0,Y 288.461,Z 332.762,A -85,B 0,C 180,E1 -17184.583,E2 -17184.583} C_VEL
LIN {X 0,Y 287.249,Z 342.478,A -85,B 0,C 180,E1 -17186.142,E2 -17186.142} C_VEL
LIN {X 0,Y 285.9,Z 351.363,A -85,B 0,C 180,E1 -17187.887,E2 -17187.887} C_VEL
LIN {X 0,Y 284.886,Z 358.679,A -85,B 0,C 180,E1 -17189.647,E2 -17189.647} C_VEL
LIN {X 0,Y 283.92,Z 365.887,A -85,B 0,C 180,E1 -17191.773,E2 -17191.773} C_VEL
LIN {X 0,Y 283.319,Z 370.75,A -85,B 0,C 180,E1 -17193.555,E2 -17193.555} C_VEL
LIN {X 0,Y 282.893,Z 375.474,A -85,B 0,C 180,E1 -17195.703,E2 -17195.703} C_VEL
LIN {X 0,Y 282.496,Z 379.102,A -85,B 0,C 180,E1 -17197.864,E2 -17197.864} C_VEL
LIN {X 0,Y 282.209,Z 381.712,A -85,B 0,C 180,E1 -17200.039,E2 -17200.039} C_VEL
LIN {X 0,Y 282.161,Z 382.935,A -85,B 0,C 180,E1 -17201.493,E2 -17201.493} C_VEL
LIN {X 0,Y 282.194,Z 383.982,A -85,B 0,C 180,E1 -17203.773,E2 -17203.773} C_VEL
LIN {X 0,Y 282.236,Z 384.047,A -85,B 0,C 180,E1 -17205.897,E2 -17205.897} C_VEL
LIN {X 0,Y 282.45,Z 383.6,A -85,B 0,C 180,E1 -17207.372,E2 -17207.372} C_VEL
LIN {X 0,Y 282.817,Z 382.415,A -85,B 0,C 180,E1 -17209.22,E2 -17209.22} C_VEL
LIN {X 0,Y 283.595,Z 379.637,A -85,B 0,C 180,E1 -17211.822,E2 -17211.822} C_VEL
LIN {X 0,Y 284.516,Z 376.266,A -85,B 0,C 180,E1 -17213.947,E2 -17213.947} C_VEL
LIN {X 0,Y 285.83,Z 371.334,A -85,B 0,C 180,E1 -17216.268,E2 -17216.268} C_VEL
LIN {X 0,Y 287.618,Z 364.65,A -85,B 0,C 180,E1 -17218.657,E2 -17218.657} C_VEL
LIN {X 0,Y 289.411,Z 357.562,A -85,B 0,C 180,E1 -17220.66,E2 -17220.66} C_VEL
LIN {X 0,Y 291.559,Z 348.872,A -85,B 0,C 180,E1 -17222.621,E2 -17222.621} C_VEL
LIN {X 0,Y 293.776,Z 338.84,A -85,B 0,C 180,E1 -17224.414,E2 -17224.414} C_VEL
LIN {X 0,Y 295.943,Z 327.89,A -85,B 0,C 180,E1 -17225.967,E2 -17225.967} C_VEL
LIN {X 0,Y 296.456,Z 323.772,A -85,B 0,C 180,E1 -17226.48,E2 -17226.48} C_VEL
LIN {X 0,Y 294.549,Z 312.243,A -85,B 0,C 180,E1 -17228.061,E2 -17228.061} C_VEL
LIN {X 0,Y 291.489,Z 300.351,A -85,B 0,C 180,E1 -17229.511,E2 -17229.511} C_VEL
LIN {X 0,Y 287.015,Z 287.445,A -85,B 0,C 180,E1 -17230.939,E2 -17230.939} C_VEL
LIN {X 0,Y 284.342,Z 281.041,A -85,B 0,C 180,E1 -17231.602,E2 -17231.602} C_VEL
LIN {X 0,Y 284.196,Z 280.207,A -85,B 0,C 180,E1 -17231.699,E2 -17231.699} C_VEL
LIN {X 0,Y 284.667,Z 276.676,A -85,B 0,C 180,E1 -17235.721,E2 -17235.721} C_VEL
LIN {X 0,Y 284.911,Z 274.579,A -85,B 0,C 180,E1 -17238.242,E2 -17238.242} C_VEL
LIN {X 0,Y 284.767,Z 271.729,A -85,B 0,C 180,E1 -17241.905,E2 -17241.905} C_VEL
LIN {X 0,Y 284.476,Z 269.236,A -85,B 0,C 180,E1 -17245.377,E2 -17245.377} C_VEL
LIN {X 0,Y 284.299,Z 268.077,A -85,B 0,C 180,E1 -17247.19,E2 -17247.19} C_VEL
LIN {X 0,Y 284.348,Z 268.069,A -85,B 0,C 180,E1 -17250.377,E2 -17250.377} C_VEL
LIN {X 0,Y 284.369,Z 268.064,A -85,B 0,C 180,E1 -17253.588,E2 -17253.588} C_VEL
LIN {X 0,Y 284.368,Z 268.061,A -85,B 0,C 180,E1 -17256.709,E2 -17256.709} C_VEL
LIN {X 0,Y 284.422,Z 268.053,A -85,B 0,C 180,E1 -17259.875,E2 -17259.875} C_VEL
LIN {X 0,Y 284.47,Z 268.05,A -85,B 0,C 180,E1 -17264.471,E2 -17264.471} C_VEL
LIN {X 0,Y 284.479,Z 268.051,A -85,B 0,C 180,E1 -17268.603,E2 -17268.603} C_VEL
LIN {X 0,Y 284.631,Z 268.03,A -85,B 0,C 180,E1 -17271.482,E2 -17271.482} C_VEL
LIN {X 0,Y 284.59,Z 268.036,A -85,B 0,C 180,E1 -17274.333,E2 -17274.333} C_VEL
LIN {X 0,Y 284.848,Z 268.004,A -85,B 0,C 180,E1 -17278.588,E2 -17278.588} C_VEL
LIN {X 0,Y 284.847,Z 268.003,A -85,B 0,C 180,E1 -17281.415,E2 -17281.415} C_VEL
LIN {X 0,Y 284.521,Z 268.043,A -85,B 0,C 180,E1 -17284.081,E2 -17284.081} C_VEL
LIN {X 0,Y 283.788,Z 268.14,A -85,B 0,C 180,E1 -17285.263,E2 -17285.263} C_VEL
LIN {X 0,Y 280.998,Z 268.493,A -85,B 0,C 180,E1 -17287.191,E2 -17287.191} C_VEL
LIN {X 0,Y 277.843,Z 268.88,A -85,B 0,C 180,E1 -17289.56,E2 -17289.56} C_VEL
LIN {X 0,Y 277.485,Z 268.92,A -85,B 0,C 180,E1 -17290.377,E2 -17290.377} C_VEL
LIN {X 0,Y 277.424,Z 268.931,A -85,B 0,C 180,E1 -17294.676,E2 -17294.676} C_VEL
LIN {X 0,Y 277.342,Z 268.942,A -85,B 0,C 180,E1 -17299.236,E2 -17299.236} C_VEL
LIN {X 0,Y 277.288,Z 268.952,A -85,B 0,C 180,E1 -17303.926,E2 -17303.926} C_VEL
LIN {X 0,Y 277.303,Z 268.949,A -85,B 0,C 180,E1 -17307.498,E2 -17307.498} C_VEL
LIN {X 0,Y 277.246,Z 268.954,A -85,B 0,C 180,E1 -17310.475,E2 -17310.475} C_VEL
LIN {X 0,Y 277.245,Z 268.951,A -85,B 0,C 180,E1 -17313.898,E2 -17313.898} C_VEL
LIN {X 0,Y 277.34,Z 269.088,A -85,B 0,C 180,E1 -17316.783,E2 -17316.783} C_VEL
LIN {X 0,Y 277.792,Z 272.083,A -85,B 0,C 180,E1 -17320.627,E2 -17320.627} C_VEL
LIN {X 0,Y 278.387,Z 275.88,A -85,B 0,C 180,E1 -17325.02,E2 -17325.02} C_VEL
LIN {X 0,Y 279.035,Z 279.746,A -85,B 0,C 180,E1 -17329.093,E2 -17329.093} C_VEL
LIN {X 0,Y 279.301,Z 281.951,A -85,B 0,C 180,E1 -17331.267,E2 -17331.267} C_VEL
LIN {X 0,Y 279.38,Z 284.482,A -85,B 0,C 180,E1 -17333.611,E2 -17333.611} C_VEL
LIN {X 0,Y 278.995,Z 287.61,A -85,B 0,C 180,E1 -17336.346,E2 -17336.346} C_VEL
LIN {X 0,Y 278.015,Z 292.852,A -85,B 0,C 180,E1 -17340.545,E2 -17340.545} C_VEL
LIN {X 0,Y 279.008,Z 296.108,A -85,B 0,C 180,E1 -17340.824,E2 -17340.824} C_VEL
LIN {X 0,Y 282.745,Z 307.94,A -85,B 0,C 180,E1 -17342.002,E2 -17342.002} C_VEL
LIN {X 0,Y 285.719,Z 320.11,A -85,B 0,C 180,E1 -17343.356,E2 -17343.356} C_VEL
LIN {X 0,Y 287.468,Z 331.593,A -85,B 0,C 180,E1 -17344.769,E2 -17344.769} C_VEL
LIN {X 0,Y 288.243,Z 342.399,A -85,B 0,C 180,E1 -17346.278,E2 -17346.278} C_VEL
LIN {X 0,Y 287.957,Z 346.193,A -85,B 0,C 180,E1 -17346.825,E2 -17346.825} C_VEL
LIN {X 0,Y 285.645,Z 356.194,A -85,B 0,C 180,E1 -17348.343,E2 -17348.343} C_VEL
LIN {X 0,Y 283.377,Z 365.249,A -85,B 0,C 180,E1 -17350.062,E2 -17350.062} C_VEL
LIN {X 0,Y 281.437,Z 373.628,A -85,B 0,C 180,E1 -17352.06,E2 -17352.06} C_VEL
LIN {X 0,Y 279.427,Z 381.234,A -85,B 0,C 180,E1 -17354.314,E2 -17354.314} C_VEL
LIN {X 0,Y 277.585,Z 387.774,A -85,B 0,C 180,E1 -17356.829,E2 -17356.829} C_VEL
LIN {X 0,Y 276.584,Z 392.125,A -85,B 0,C 180,E1 -17359.014,E2 -17359.014} C_VEL
LIN {X 0,Y 275.858,Z 395.43,A -85,B 0,C 180,E1 -17361.208,E2 -17361.208} C_VEL
LIN {X 0,Y 275.307,Z 398.349,A -85,B 0,C 180,E1 -17364.139,E2 -17364.139} C_VEL
LIN {X 0,Y 275.232,Z 399.213,A -85,B 0,C 180,E1 -17365.607,E2 -17365.607} C_VEL
LIN {X 0,Y 275.248,Z 399.65,A -85,B 0,C 180,E1 -17367.073,E2 -17367.073} C_VEL
LIN {X 0,Y 275.258,Z 399.7,A -85,B 0,C 180,E1 -17368.537,E2 -17368.537} C_VEL
LIN {X 0,Y 275.28,Z 399.366,A -85,B 0,C 180,E1 -17370,E2 -17370} C_VEL
LIN {X 0,Y 275.271,Z 398.64,A -85,B 0,C 180,E1 -17371.463,E2 -17371.463} C_VEL
LIN {X 0,Y 275.283,Z 397.468,A -85,B 0,C 180,E1 -17372.927,E2 -17372.927} C_VEL
LIN {X 0,Y 275.324,Z 394.523,A -85,B 0,C 180,E1 -17375.409,E2 -17375.409} C_VEL
LIN {X 0,Y 275.599,Z 389.939,A -85,B 0,C 180,E1 -17378.062,E2 -17378.062} C_VEL
LIN {X 0,Y 276.095,Z 384.865,A -85,B 0,C 180,E1 -17380.264,E2 -17380.264} C_VEL
LIN {X 0,Y 276.82,Z 378.463,A -85,B 0,C 180,E1 -17382.462,E2 -17382.462} C_VEL
LIN {X 0,Y 277.984,Z 370.44,A -85,B 0,C 180,E1 -17384.644,E2 -17384.644} C_VEL
LIN {X 0,Y 279.199,Z 361.651,A -85,B 0,C 180,E1 -17386.574,E2 -17386.574} C_VEL
LIN {X 0,Y 280.418,Z 352.225,A -85,B 0,C 180,E1 -17388.257,E2 -17388.257} C_VEL
LIN {X 0,Y 281.751,Z 342.362,A -85,B 0,C 180,E1 -17389.678,E2 -17389.678} C_VEL
LIN {X 0,Y 282.273,Z 338.055,A -85,B 0,C 180,E1 -17390.209,E2 -17390.209} C_VEL
LIN {X 0,Y 281.445,Z 326.962,A -85,B 0,C 180,E1 -17391.489,E2 -17391.489} C_VEL
LIN {X 0,Y 280.036,Z 314.31,A -85,B 0,C 180,E1 -17392.654,E2 -17392.654} C_VEL
LIN {X 0,Y 277.981,Z 301.184,A -85,B 0,C 180,E1 -17393.595,E2 -17393.595} C_VEL
LIN {X 0,Y 276.466,Z 293.345,A -85,B 0,C 180,E1 -17394.049,E2 -17394.049} C_VEL
LIN {X 0,Y 276.924,Z 288.933,A -85,B 0,C 180,E1 -17397.342,E2 -17397.342} C_VEL
LIN {X 0,Y 277.863,Z 282.69,A -85,B 0,C 180,E1 -17402.083,E2 -17402.083} C_VEL
LIN {X 0,Y 278.466,Z 278.366,A -85,B 0,C 180,E1 -17405.483,E2 -17405.483} C_VEL
LIN {X 0,Y 278.509,Z 276.16,A -85,B 0,C 180,E1 -17407.273,E2 -17407.273} C_VEL
LIN {X 0,Y 277.777,Z 271.727,A -85,B 0,C 180,E1 -17411.133,E2 -17411.133} C_VEL
LIN {X 0,Y 277.258,Z 268.95,A -85,B 0,C 180,E1 -17413.768,E2 -17413.768} C_VEL
LIN {X 0,Y 277.188,Z 268.96,A -85,B 0,C 180,E1 -17417.33,E2 -17417.33} C_VEL
LIN {X 0,Y 277.247,Z 268.95,A -85,B 0,C 180,E1 -17421.796,E2 -17421.796} C_VEL
LIN {X 0,Y 277.275,Z 268.947,A -85,B 0,C 180,E1 -17424.338,E2 -17424.338} C_VEL
LIN {X 0,Y 277.238,Z 268.949,A -85,B 0,C 180,E1 -17427.834,E2 -17427.834} C_VEL
LIN {X 0,Y 277.237,Z 268.949,A -85,B 0,C 180,E1 -17431.205,E2 -17431.205} C_VEL
LIN {X 0,Y 277.244,Z 268.952,A -85,B 0,C 180,E1 -17434.471,E2 -17434.471} C_VEL
LIN {X 0,Y 277.259,Z 268.946,A -85,B 0,C 180,E1 -17437.651,E2 -17437.651} C_VEL
LIN {X 0,Y 277.339,Z 268.937,A -85,B 0,C 180,E1 -17440.764,E2 -17440.764} C_VEL
LIN {X 0,Y 277.424,Z 268.926,A -85,B 0,C 180,E1 -17445.324,E2 -17445.324} C_VEL
LIN {X 0,Y 277.457,Z 268.921,A -85,B 0,C 180,E1 -17449.785,E2 -17449.785} C_VEL
LIN {X 0,Y 277.636,Z 268.9,A -85,B 0,C 180,E1 -17452.727,E2 -17452.727} C_VEL
LIN {X 0,Y 277.816,Z 268.865,A -85,B 0,C 180,E1 -17458.549,E2 -17458.549} C_VEL
LIN {X 0,Y 277.816,Z 268.871,A -85,B 0,C 180,E1 -17461.448,E2 -17461.448} C_VEL
LIN {X 0,Y 277.646,Z 268.9,A -85,B 0,C 180,E1 -17467.269,E2 -17467.269} C_VEL
LIN {X 0,Y 277.499,Z 268.915,A -85,B 0,C 180,E1 -17470.21,E2 -17470.21} C_VEL
LIN {X 0,Y 277.42,Z 268.926,A -85,B 0,C 180,E1 -17474.673,E2 -17474.673} C_VEL
LIN {X 0,Y 277.336,Z 268.938,A -85,B 0,C 180,E1 -17479.232,E2 -17479.232} C_VEL
LIN {X 0,Y 277.31,Z 268.937,A -85,B 0,C 180,E1 -17484.169,E2 -17484.169} C_VEL
LIN {X 0,Y 277.317,Z 268.941,A -85,B 0,C 180,E1 -17487.504,E2 -17487.504} C_VEL
LIN {X 0,Y 277.263,Z 268.942,A -85,B 0,C 180,E1 -17490.48,E2 -17490.48} C_VEL
LIN {X 0,Y 277.244,Z 268.947,A -85,B 0,C 180,E1 -17493.894,E2 -17493.894} C_VEL
LIN {X 0,Y 277.276,Z 268.944,A -85,B 0,C 180,E1 -17497.465,E2 -17497.465} C_VEL
LIN {X 0,Y 277.282,Z 268.943,A -85,B 0,C 180,E1 -17501.221,E2 -17501.221} C_VEL
LIN {X 0,Y 277.232,Z 268.951,A -85,B 0,C 180,E1 -17505.217,E2 -17505.217} C_VEL
LIN {X 0,Y 277.215,Z 268.952,A -85,B 0,C 180,E1 -17509.511,E2 -17509.511} C_VEL
LIN {X 0,Y 277.266,Z 268.948,A -85,B 0,C 180,E1 -17512.531,E2 -17512.531} C_VEL
LIN {X 0,Y 277.243,Z 268.95,A -85,B 0,C 180,E1 -17516.105,E2 -17516.105} C_VEL
LIN {X 0,Y 277.251,Z 268.947,A -85,B 0,C 180,E1 -17519.538,E2 -17519.538} C_VEL
LIN {X 0,Y 277.328,Z 268.939,A -85,B 0,C 180,E1 -17522.861,E2 -17522.861} C_VEL
LIN {X 0,Y 277.196,Z 268.958,A -85,B 0,C 180,E1 -17527.746,E2 -17527.746} C_VEL
LIN {X 0,Y 276.943,Z 271.656,A -85,B 0,C 180,E1 -17530.738,E2 -17530.738} C_VEL
LIN {X 0,Y 276.658,Z 276,A -85,B 0,C 180,E1 -17535.284,E2 -17535.284} C_VEL
LIN {X 0,Y 276.338,Z 279.743,A -85,B 0,C 180,E1 -17539.051,E2 -17539.051} C_VEL
LIN {X 0,Y 279.746,Z 293.483,A -85,B 0,C 180,E1 -17539.988,E2 -17539.988} C_VEL
LIN {X 0,Y 281.901,Z 305.157,A -85,B 0,C 180,E1 -17540.991,E2 -17540.991} C_VEL
LIN {X 0,Y 283.368,Z 316.304,A -85,B 0,C 180,E1 -17542.16,E2 -17542.16} C_VEL
LIN {X 0,Y 283.106,Z 321.066,A -85,B 0,C 180,E1 -17542.691,E2 -17542.691} C_VEL
LIN {X 0,Y 281.683,Z 332.056,A -85,B 0,C 180,E1 -17544.093,E2 -17544.093} C_VEL
LIN {X 0,Y 280.402,Z 341.931,A -85,B 0,C 180,E1 -17545.688,E2 -17545.688} C_VEL
LIN {X 0,Y 279.02,Z 350.936,A -85,B 0,C 180,E1 -17547.474,E2 -17547.474} C_VEL
LIN {X 0,Y 278.001,Z 358.349,A -85,B 0,C 180,E1 -17549.276,E2 -17549.276} C_VEL
LIN {X 0,Y 276.924,Z 365.658,A -85,B 0,C 180,E1 -17551.454,E2 -17551.454} C_VEL
LIN {X 0,Y 276.191,Z 371.508,A -85,B 0,C 180,E1 -17553.647,E2 -17553.647} C_VEL
LIN {X 0,Y 275.719,Z 376.797,A -85,B 0,C 180,E1 -17556.249,E2 -17556.249} C_VEL
LIN {X 0,Y 275.253,Z 380.555,A -85,B 0,C 180,E1 -17558.812,E2 -17558.812} C_VEL
LIN {X 0,Y 275.09,Z 382.141,A -85,B 0,C 180,E1 -17560.302,E2 -17560.302} C_VEL
LIN {X 0,Y 275.072,Z 383.27,A -85,B 0,C 180,E1 -17561.794,E2 -17561.794} C_VEL
LIN {X 0,Y 275.11,Z 384.183,A -85,B 0,C 180,E1 -17563.901,E2 -17563.901} C_VEL
LIN {X 0,Y 275.201,Z 384.22,A -85,B 0,C 180,E1 -17566.314,E2 -17566.314} C_VEL
LIN {X 0,Y 275.433,Z 383.678,A -85,B 0,C 180,E1 -17567.83,E2 -17567.83} C_VEL
LIN {X 0,Y 275.78,Z 382.641,A -85,B 0,C 180,E1 -17569.46,E2 -17569.46} C_VEL
LIN {X 0,Y 276.208,Z 381.359,A -85,B 0,C 180,E1 -17570.868,E2 -17570.868} C_VEL
LIN {X 0,Y 277.04,Z 378.422,A -85,B 0,C 180,E1 -17573.154,E2 -17573.154} C_VEL
LIN {X 0,Y 278.206,Z 374.376,A -85,B 0,C 180,E1 -17575.432,E2 -17575.432} C_VEL
LIN {X 0,Y 280.013,Z 368.037,A -85,B 0,C 180,E1 -17578.073,E2 -17578.073} C_VEL
LIN {X 0,Y 281.897,Z 361.043,A -85,B 0,C 180,E1 -17580.321,E2 -17580.321} C_VEL
LIN {X 0,Y 283.834,Z 353.849,A -85,B 0,C 180,E1 -17582.164,E2 -17582.164} C_VEL
LIN {X 0,Y 286.012,Z 345.092,A -85,B 0,C 180,E1 -17583.987,E2 -17583.987} C_VEL
LIN {X 0,Y 288.187,Z 335.363,A -85,B 0,C 180,E1 -17585.607,E2 -17585.607} C_VEL
LIN {X 0,Y 290.014,Z 325.8,A -85,B 0,C 180,E1 -17586.902,E2 -17586.902} C_VEL
LIN {X 0,Y 288.288,Z 314.619,A -85,B 0,C 180,E1 -17588.523,E2 -17588.523} C_VEL
LIN {X 0,Y 285.685,Z 303.928,A -85,B 0,C 180,E1 -17589.927,E2 -17589.927} C_VEL
LIN {X 0,Y 281.512,Z 291.253,A -85,B 0,C 180,E1 -17591.444,E2 -17591.444} C_VEL
LIN {X 0,Y 277.416,Z 281.223,A -85,B 0,C 180,E1 -17592.548,E2 -17592.548} C_VEL
LIN {X 0,Y 277.275,Z 280.431,A -85,B 0,C 180,E1 -17592.648,E2 -17592.648} C_VEL
LIN {X 0,Y 277.772,Z 276.825,A -85,B 0,C 180,E1 -17596.914,E2 -17596.914} C_VEL
LIN {X 0,Y 277.868,Z 274.898,A -85,B 0,C 180,E1 -17599.355,E2 -17599.355} C_VEL
LIN {X 0,Y 277.726,Z 272.49,A -85,B 0,C 180,E1 -17602.606,E2 -17602.606} C_VEL
LIN {X 0,Y 277.361,Z 269.644,A -85,B 0,C 180,E1 -17606.737,E2 -17606.737} C_VEL
LIN {X 0,Y 277.235,Z 268.956,A -85,B 0,C 180,E1 -17607.838,E2 -17607.838} C_VEL
LIN {X 0,Y 277.261,Z 268.948,A -85,B 0,C 180,E1 -17611.212,E2 -17611.212} C_VEL
LIN {X 0,Y 277.31,Z 268.941,A -85,B 0,C 180,E1 -17614.481,E2 -17614.481} C_VEL
LIN {X 0,Y 277.29,Z 268.943,A -85,B 0,C 180,E1 -17617.657,E2 -17617.657} C_VEL
LIN {X 0,Y 277.363,Z 268.937,A -85,B 0,C 180,E1 -17620.77,E2 -17620.77} C_VEL
LIN {X 0,Y 277.42,Z 268.923,A -85,B 0,C 180,E1 -17625.327,E2 -17625.327} C_VEL
LIN {X 0,Y 277.453,Z 268.924,A -85,B 0,C 180,E1 -17629.789,E2 -17629.789} C_VEL
LIN {X 0,Y 277.633,Z 268.904,A -85,B 0,C 180,E1 -17632.73,E2 -17632.73} C_VEL
LIN {X 0,Y 277.814,Z 268.88,A -85,B 0,C 180,E1 -17638.552,E2 -17638.552} C_VEL
LIN {X 0,Y 277.813,Z 268.879,A -85,B 0,C 180,E1 -17641.451,E2 -17641.451} C_VEL
LIN {X 0,Y 277.647,Z 268.9,A -85,B 0,C 180,E1 -17647.273,E2 -17647.273} C_VEL
LIN {X 0,Y 277.485,Z 268.92,A -85,B 0,C 180,E1 -17650.377,E2 -17650.377} C_VEL
LIN {X 0,Y 276.754,Z 269.012,A -85,B 0,C 180,E1 -17651.587,E2 -17651.587} C_VEL
LIN {X 0,Y 273.912,Z 269.367,A -85,B 0,C 180,E1 -17653.56,E2 -17653.56} C_VEL
LIN {X 0,Y 271.513,Z 269.671,A -85,B 0,C 180,E1 -17655.162,E2 -17655.162} C_VEL
LIN {X 0,Y 270.442,Z 269.803,A -85,B 0,C 180,E1 -17656.402,E2 -17656.402} C_VEL
LIN {X 0,Y 270.329,Z 269.815,A -85,B 0,C 180,E1 -17656.823,E2 -17656.823} C_VEL
LIN {X 0,Y 270.289,Z 269.822,A -85,B 0,C 180,E1 -17660.603,E2 -17660.603} C_VEL
LIN {X 0,Y 270.231,Z 269.83,A -85,B 0,C 180,E1 -17664.591,E2 -17664.591} C_VEL
LIN {X 0,Y 270.24,Z 269.828,A -85,B 0,C 180,E1 -17667.914,E2 -17667.914} C_VEL
LIN {X 0,Y 270.172,Z 269.836,A -85,B 0,C 180,E1 -17671.351,E2 -17671.351} C_VEL
LIN {X 0,Y 270.247,Z 269.867,A -85,B 0,C 180,E1 -17675.69,E2 -17675.69} C_VEL
LIN {X 0,Y 270.655,Z 272.16,A -85,B 0,C 180,E1 -17678.833,E2 -17678.833} C_VEL
LIN {X 0,Y 271.049,Z 275.004,A -85,B 0,C 180,E1 -17682.39,E2 -17682.39} C_VEL
LIN {X 0,Y 271.612,Z 278.53,A -85,B 0,C 180,E1 -17686.43,E2 -17686.43} C_VEL
LIN {X 0,Y 272.121,Z 281.723,A -85,B 0,C 180,E1 -17689.785,E2 -17689.785} C_VEL
LIN {X 0,Y 272.376,Z 285.113,A -85,B 0,C 180,E1 -17693.121,E2 -17693.121} C_VEL
LIN {X 0,Y 272.047,Z 288.036,A -85,B 0,C 180,E1 -17695.761,E2 -17695.761} C_VEL
LIN {X 0,Y 271.179,Z 292.423,A -85,B 0,C 180,E1 -17699.532,E2 -17699.532} C_VEL
LIN {X 0,Y 272.117,Z 295.756,A -85,B 0,C 180,E1 -17699.836,E2 -17699.836} C_VEL
LIN {X 0,Y 275.997,Z 307.491,A -85,B 0,C 180,E1 -17701.081,E2 -17701.081} C_VEL
LIN {X 0,Y 278.894,Z 319.213,A -85,B 0,C 180,E1 -17702.435,E2 -17702.435} C_VEL
LIN {X 0,Y 280.708,Z 330.007,A -85,B 0,C 180,E1 -17703.813,E2 -17703.813} C_VEL
LIN {X 0,Y 281.658,Z 341.762,A -85,B 0,C 180,E1 -17705.492,E2 -17705.492} C_VEL
LIN {X 0,Y 281.474,Z 346.778,A -85,B 0,C 180,E1 -17706.259,E2 -17706.259} C_VEL
LIN {X 0,Y 279.087,Z 356.609,A -85,B 0,C 180,E1 -17707.807,E2 -17707.807} C_VEL
LIN {X 0,Y 276.733,Z 365.563,A -85,B 0,C 180,E1 -17709.562,E2 -17709.562} C_VEL
LIN {X 0,Y 274.943,Z 372.508,A -85,B 0,C 180,E1 -17711.234,E2 -17711.234} C_VEL
LIN {X 0,Y 272.939,Z 380.274,A -85,B 0,C 180,E1 -17713.547,E2 -17713.547} C_VEL
LIN {X 0,Y 271.149,Z 386.161,A -85,B 0,C 180,E1 -17715.746,E2 -17715.746} C_VEL
LIN {X 0,Y 269.928,Z 390.825,A -85,B 0,C 180,E1 -17717.978,E2 -17717.978} C_VEL
LIN {X 0,Y 269.041,Z 394.405,A -85,B 0,C 180,E1 -17720.224,E2 -17720.224} C_VEL
LIN {X 0,Y 268.481,Z 397,A -85,B 0,C 180,E1 -17722.48,E2 -17722.48} C_VEL
LIN {X 0,Y 268.207,Z 398.666,A -85,B 0,C 180,E1 -17724.721,E2 -17724.721} C_VEL
LIN {X 0,Y 268.16,Z 399.461,A -85,B 0,C 180,E1 -17726.996,E2 -17726.996} C_VEL
LIN {X 0,Y 268.184,Z 399.488,A -85,B 0,C 180,E1 -17728.498,E2 -17728.498} C_VEL
LIN {X 0,Y 268.204,Z 399.13,A -85,B 0,C 180,E1 -17730,E2 -17730} C_VEL
LIN {X 0,Y 268.198,Z 398.364,A -85,B 0,C 180,E1 -17731.502,E2 -17731.502} C_VEL
LIN {X 0,Y 268.194,Z 397.157,A -85,B 0,C 180,E1 -17733.004,E2 -17733.004} C_VEL
LIN {X 0,Y 268.216,Z 394.519,A -85,B 0,C 180,E1 -17735.299,E2 -17735.299} C_VEL
LIN {X 0,Y 268.427,Z 390.959,A -85,B 0,C 180,E1 -17737.522,E2 -17737.522} C_VEL
LIN {X 0,Y 268.873,Z 386.214,A -85,B 0,C 180,E1 -17739.782,E2 -17739.782} C_VEL
LIN {X 0,Y 269.683,Z 379.06,A -85,B 0,C 180,E1 -17742.415,E2 -17742.415} C_VEL
LIN {X 0,Y 270.875,Z 371.277,A -85,B 0,C 180,E1 -17744.653,E2 -17744.653} C_VEL
LIN {X 0,Y 272.206,Z 361.879,A -85,B 0,C 180,E1 -17746.8,E2 -17746.8} C_VEL
LIN {X 0,Y 273.608,Z 351.327,A -85,B 0,C 180,E1 -17748.728,E2 -17748.728} C_VEL
LIN {X 0,Y 275.227,Z 339.828,A -85,B 0,C 180,E1 -17750.36,E2 -17750.36} C_VEL
LIN {X 0,Y 274.71,Z 329.808,A -85,B 0,C 180,E1 -17751.595,E2 -17751.595} C_VEL
LIN {X 0,Y 273.541,Z 317.866,A -85,B 0,C 180,E1 -17752.807,E2 -17752.807} C_VEL
LIN {X 0,Y 271.718,Z 305.003,A -85,B 0,C 180,E1 -17753.836,E2 -17753.836} C_VEL
LIN {X 0,Y 269.431,Z 293.157,A -85,B 0,C 180,E1 -17754.572,E2 -17754.572} C_VEL
LIN {X 0,Y 270.063,Z 287.701,A -85,B 0,C 180,E1 -17758.779,E2 -17758.779} C_VEL
LIN {X 0,Y 270.95,Z 282.315,A -85,B 0,C 180,E1 -17763.004,E2 -17763.004} C_VEL
LIN {X 0,Y 271.448,Z 279.084,A -85,B 0,C 180,E1 -17765.629,E2 -17765.629} C_VEL
LIN {X 0,Y 271.324,Z 275.796,A -85,B 0,C 180,E1 -17768.437,E2 -17768.437} C_VEL
LIN {X 0,Y 270.524,Z 271.316,A -85,B 0,C 180,E1 -17772.489,E2 -17772.489} C_VEL
LIN {X 0,Y 270.211,Z 269.828,A -85,B 0,C 180,E1 -17774.008,E2 -17774.008} C_VEL
LIN {X 0,Y 270.148,Z 269.837,A -85,B 0,C 180,E1 -17777.435,E2 -17777.435} C_VEL
LIN {X 0,Y 270.177,Z 269.832,A -85,B 0,C 180,E1 -17781.367,E2 -17781.367} C_VEL
LIN {X 0,Y 270.196,Z 269.828,A -85,B 0,C 180,E1 -17785.092,E2 -17785.092} C_VEL
LIN {X 0,Y 270.183,Z 269.827,A -85,B 0,C 180,E1 -17789.135,E2 -17789.135} C_VEL
LIN {X 0,Y 270.221,Z 269.824,A -85,B 0,C 180,E1 -17792.161,E2 -17792.161} C_VEL
LIN {X 0,Y 270.225,Z 269.821,A -85,B 0,C 180,E1 -17795.541,E2 -17795.541} C_VEL
LIN {X 0,Y 270.297,Z 269.818,A -85,B 0,C 180,E1 -17800.242,E2 -17800.242} C_VEL
LIN {X 0,Y 270.393,Z 269.803,A -85,B 0,C 180,E1 -17804.933,E2 -17804.933} C_VEL
LIN {X 0,Y 270.409,Z 269.798,A -85,B 0,C 180,E1 -17809.516,E2 -17809.516} C_VEL
LIN {X 0,Y 270.594,Z 269.778,A -85,B 0,C 180,E1 -17812.537,E2 -17812.537} C_VEL
LIN {X 0,Y 270.782,Z 269.74,A -85,B 0,C 180,E1 -17818.511,E2 -17818.511} C_VEL
LIN {X 0,Y 270.782,Z 269.746,A -85,B 0,C 180,E1 -17821.485,E2 -17821.485} C_VEL
LIN {X 0,Y 270.604,Z 269.778,A -85,B 0,C 180,E1 -17827.459,E2 -17827.459} C_VEL
LIN {X 0,Y 270.435,Z 269.794,A -85,B 0,C 180,E1 -17830.479,E2 -17830.479} C_VEL
LIN {X 0,Y 270.389,Z 269.803,A -85,B 0,C 180,E1 -17835.063,E2 -17835.063} C_VEL
LIN {X 0,Y 270.293,Z 269.816,A -85,B 0,C 180,E1 -17839.754,E2 -17839.754} C_VEL
LIN {X 0,Y 270.266,Z 269.814,A -85,B 0,C 180,E1 -17844.584,E2 -17844.584} C_VEL
LIN {X 0,Y 270.263,Z 269.817,A -85,B 0,C 180,E1 -17847.907,E2 -17847.907} C_VEL
LIN {X 0,Y 270.175,Z 269.83,A -85,B 0,C 180,E1 -17851.347,E2 -17851.347} C_VEL
LIN {X 0,Y 270.205,Z 269.827,A -85,B 0,C 180,E1 -17854.902,E2 -17854.902} C_VEL
LIN {X 0,Y 270.213,Z 269.825,A -85,B 0,C 180,E1 -17858.716,E2 -17858.716} C_VEL
LIN {X 0,Y 270.237,Z 269.82,A -85,B 0,C 180,E1 -17862.543,E2 -17862.543} C_VEL
LIN {X 0,Y 270.179,Z 269.83,A -85,B 0,C 180,E1 -17866.745,E2 -17866.745} C_VEL
LIN {X 0,Y 270.197,Z 269.826,A -85,B 0,C 180,E1 -17871.373,E2 -17871.373} C_VEL
LIN {X 0,Y 270.204,Z 269.826,A -85,B 0,C 180,E1 -17875.096,E2 -17875.096} C_VEL
LIN {X 0,Y 270.19,Z 269.828,A -85,B 0,C 180,E1 -17879.13,E2 -17879.13} C_VEL
LIN {X 0,Y 270.249,Z 269.822,A -85,B 0,C 180,E1 -17882.147,E2 -17882.147} C_VEL
LIN {X 0,Y 270.157,Z 269.833,A -85,B 0,C 180,E1 -17885.57,E2 -17885.57} C_VEL
LIN {X 0,Y 270.187,Z 269.943,A -85,B 0,C 180,E1 -17887.842,E2 -17887.842} C_VEL
LIN {X 0,Y 269.784,Z 273.53,A -85,B 0,C 180,E1 -17891.784,E2 -17891.784} C_VEL
LIN {X 0,Y 269.647,Z 276.42,A -85,B 0,C 180,E1 -17894.892,E2 -17894.892} C_VEL
LIN {X 0,Y 269.32,Z 279.926,A -85,B 0,C 180,E1 -17898.524,E2 -17898.524} C_VEL
LIN {X 0,Y 272.665,Z 293.438,A -85,B 0,C 180,E1 -17899.472,E2 -17899.472} C_VEL
LIN {X 0,Y 274.792,Z 304.507,A -85,B 0,C 180,E1 -17900.448,E2 -17900.448} C_VEL
LIN {X 0,Y 276.314,Z 315.226,A -85,B 0,C 180,E1 -17901.59,E2 -17901.59} C_VEL
LIN {X 0,Y 276.449,Z 319.997,A -85,B 0,C 180,E1 -17902.146,E2 -17902.146} C_VEL
LIN {X 0,Y 274.929,Z 331.253,A -85,B 0,C 180,E1 -17903.579,E2 -17903.579} C_VEL
LIN {X 0,Y 273.571,Z 341.355,A -85,B 0,C 180,E1 -17905.211,E2 -17905.211} C_VEL
LIN {X 0,Y 272.183,Z 350.479,A -85,B 0,C 180,E1 -17907.04,E2 -17907.04} C_VEL
LIN {X 0,Y 270.852,Z 359.369,A -85,B 0,C 180,E1 -17909.257,E2 -17909.257} C_VEL
LIN {X 0,Y 269.833,Z 366.516,A -85,B 0,C 180,E1 -17911.492,E2 -17911.492} C_VEL
LIN {X 0,Y 269.071,Z 372.214,A -85,B 0,C 180,E1 -17913.744,E2 -17913.744} C_VEL
LIN {X 0,Y 268.638,Z 377.064,A -85,B 0,C 180,E1 -17916.227,E2 -17916.227} C_VEL
LIN {X 0,Y 268.124,Z 381.031,A -85,B 0,C 180,E1 -17919.048,E2 -17919.048} C_VEL
LIN {X 0,Y 267.975,Z 382.541,A -85,B 0,C 180,E1 -17920.578,E2 -17920.578} C_VEL
LIN {X 0,Y 267.975,Z 383.596,A -85,B 0,C 180,E1 -17922.111,E2 -17922.111} C_VEL
LIN {X 0,Y 268.007,Z 384.378,A -85,B 0,C 180,E1 -17924.018,E2 -17924.018} C_VEL
LIN {X 0,Y 268.152,Z 384.356,A -85,B 0,C 180,E1 -17926.756,E2 -17926.756} C_VEL
LIN {X 0,Y 268.744,Z 382.872,A -85,B 0,C 180,E1 -17929.711,E2 -17929.711} C_VEL
LIN {X 0,Y 269.302,Z 381.318,A -85,B 0,C 180,E1 -17931.429,E2 -17931.429} C_VEL
LIN {X 0,Y 270.238,Z 378.274,A -85,B 0,C 180,E1 -17933.772,E2 -17933.772} C_VEL
LIN {X 0,Y 271.505,Z 374.096,A -85,B 0,C 180,E1 -17936.106,E2 -17936.106} C_VEL
LIN {X 0,Y 273.459,Z 367.61,A -85,B 0,C 180,E1 -17938.808,E2 -17938.808} C_VEL
LIN {X 0,Y 275.524,Z 360.471,A -85,B 0,C 180,E1 -17941.099,E2 -17941.099} C_VEL
LIN {X 0,Y 277.481,Z 353.417,A -85,B 0,C 180,E1 -17942.908,E2 -17942.908} C_VEL
LIN {X 0,Y 279.88,Z 344.074,A -85,B 0,C 180,E1 -17944.838,E2 -17944.838} C_VEL
LIN {X 0,Y 282.178,Z 334.098,A -85,B 0,C 180,E1 -17946.486,E2 -17946.486} C_VEL
LIN {X 0,Y 283.504,Z 327.739,A -85,B 0,C 180,E1 -17947.366,E2 -17947.366} C_VEL
LIN {X 0,Y 282.197,Z 317.914,A -85,B 0,C 180,E1 -17948.876,E2 -17948.876} C_VEL
LIN {X 0,Y 279.556,Z 306.303,A -85,B 0,C 180,E1 -17950.497,E2 -17950.497} C_VEL
LIN {X 0,Y 275.654,Z 294.148,A -85,B 0,C 180,E1 -17952.053,E2 -17952.053} C_VEL
LIN {X 0,Y 271.386,Z 283.783,A -85,B 0,C 180,E1 -17953.305,E2 -17953.305} C_VEL
LIN {X 0,Y 270.35,Z 280.678,A -85,B 0,C 180,E1 -17953.638,E2 -17953.638} C_VEL
LIN {X 0,Y 270.801,Z 277.47,A -85,B 0,C 180,E1 -17957.567,E2 -17957.567} C_VEL
LIN {X 0,Y 270.808,Z 274.803,A -85,B 0,C 180,E1 -17961.127,E2 -17961.127} C_VEL
LIN {X 0,Y 270.496,Z 272.027,A -85,B 0,C 180,E1 -17965.141,E2 -17965.141} C_VEL
LIN {X 0,Y 270.175,Z 269.835,A -85,B 0,C 180,E1 -17968.653,E2 -17968.653} C_VEL
LIN {X 0,Y 270.255,Z 269.822,A -85,B 0,C 180,E1 -17972.147,E2 -17972.147} C_VEL
LIN {X 0,Y 270.273,Z 269.819,A -85,B 0,C 180,E1 -17975.518,E2 -17975.518} C_VEL
LIN {X 0,Y 270.318,Z 269.811,A -85,B 0,C 180,E1 -17980.248,E2 -17980.248} C_VEL
LIN {X 0,Y 270.388,Z 269.8,A -85,B 0,C 180,E1 -17984.937,E2 -17984.937} C_VEL
LIN {X 0,Y 270.405,Z 269.803,A -85,B 0,C 180,E1 -17989.519,E2 -17989.519} C_VEL
LIN {X 0,Y 270.591,Z 269.78,A -85,B 0,C 180,E1 -17992.54,E2 -17992.54} C_VEL
LIN {X 0,Y 270.78,Z 269.756,A -85,B 0,C 180,E1 -17998.515,E2 -17998.515} C_VEL
LIN {X 0,Y 270.78,Z 269.755,A -85,B 0,C 180,E1 -18001.489,E2 -18001.489} C_VEL
LIN {X 0,Y 270.605,Z 269.777,A -85,B 0,C 180,E1 -18007.463,E2 -18007.463} C_VEL
LIN {X 0,Y 270.437,Z 269.799,A -85,B 0,C 180,E1 -18010.483,E2 -18010.483} C_VEL
LIN {X 0,Y 270.392,Z 269.807,A -85,B 0,C 180,E1 -18015.067,E2 -18015.067} C_VEL
LIN {X 0,Y 270.329,Z 269.815,A -85,B 0,C 180,E1 -18016.823,E2 -18016.823} C_VEL
LIN {X 0,Y 269.572,Z 269.911,A -85,B 0,C 180,E1 -18018.066,E2 -18018.066} C_VEL
LIN {X 0,Y 266.625,Z 270.281,A -85,B 0,C 180,E1 -18020.09,E2 -18020.09} C_VEL
LIN {X 0,Y 264.196,Z 270.583,A -85,B 0,C 180,E1 -18021.737,E2 -18021.737} C_VEL
LIN {X 0,Y 263.199,Z 270.706,A -85,B 0,C 180,E1 -18023.014,E2 -18023.014} C_VEL
LIN {X 0,Y 263.14,Z 270.714,A -85,B 0,C 180,E1 -18023.447,E2 -18023.447} C_VEL
LIN {X 0,Y 263.177,Z 270.71,A -85,B 0,C 180,E1 -18027.001,E2 -18027.001} C_VEL
LIN {X 0,Y 263.128,Z 270.713,A -85,B 0,C 180,E1 -18031.276,E2 -18031.276} C_VEL
LIN {X 0,Y 263.151,Z 270.708,A -85,B 0,C 180,E1 -18034.116,E2 -18034.116} C_VEL
LIN {X 0,Y 263.479,Z 272.22,A -85,B 0,C 180,E1 -18036.851,E2 -18036.851} C_VEL
LIN {X 0,Y 263.788,Z 274.359,A -85,B 0,C 180,E1 -18039.751,E2 -18039.751} C_VEL
LIN {X 0,Y 264.271,Z 277.561,A -85,B 0,C 180,E1 -18043.746,E2 -18043.746} C_VEL
LIN {X 0,Y 264.895,Z 281.271,A -85,B 0,C 180,E1 -18047.979,E2 -18047.979} C_VEL
LIN {X 0,Y 265.206,Z 283.677,A -85,B 0,C 180,E1 -18050.507,E2 -18050.507} C_VEL
LIN {X 0,Y 265.345,Z 285.782,A -85,B 0,C 180,E1 -18052.619,E2 -18052.619} C_VEL
LIN {X 0,Y 265.086,Z 288.606,A -85,B 0,C 180,E1 -18055.275,E2 -18055.275} C_VEL
LIN {X 0,Y 264.342,Z 292.205,A -85,B 0,C 180,E1 -18058.469,E2 -18058.469} C_VEL
LIN {X 0,Y 265.529,Z 295.899,A -85,B 0,C 180,E1 -18058.851,E2 -18058.851} C_VEL
LIN {X 0,Y 269.721,Z 308.856,A -85,B 0,C 180,E1 -18060.305,E2 -18060.305} C_VEL
LIN {X 0,Y 272.829,Z 321.918,A -85,B 0,C 180,E1 -18061.918,E2 -18061.918} C_VEL
LIN {X 0,Y 274.485,Z 333.208,A -85,B 0,C 180,E1 -18063.467,E2 -18063.467} C_VEL
LIN {X 0,Y 275.131,Z 343.688,A -85,B 0,C 180,E1 -18065.073,E2 -18065.073} C_VEL
LIN {X 0,Y 275.021,Z 347.348,A -85,B 0,C 180,E1 -18065.666,E2 -18065.666} C_VEL
LIN {X 0,Y 272.558,Z 357.042,A -85,B 0,C 180,E1 -18067.246,E2 -18067.246} C_VEL
LIN {X 0,Y 270.098,Z 365.887,A -85,B 0,C 180,E1 -18069.037,E2 -18069.037} C_VEL
LIN {X 0,Y 267.817,Z 374.535,A -85,B 0,C 180,E1 -18071.247,E2 -18071.247} C_VEL
LIN {X 0,Y 265.797,Z 381.487,A -85,B 0,C 180,E1 -18073.487,E2 -18073.487} C_VEL
LIN {X 0,Y 263.728,Z 387.884,A -85,B 0,C 180,E1 -18076.123,E2 -18076.123} C_VEL
LIN {X 0,Y 262.615,Z 392.116,A -85,B 0,C 180,E1 -18078.422,E2 -18078.422} C_VEL
LIN {X 0,Y 261.793,Z 395.311,A -85,B 0,C 180,E1 -18080.731,E2 -18080.731} C_VEL
LIN {X 0,Y 261.161,Z 398.118,A -85,B 0,C 180,E1 -18083.821,E2 -18083.821} C_VEL
LIN {X 0,Y 261.072,Z 398.889,A -85,B 0,C 180,E1 -18085.368,E2 -18085.368} C_VEL
LIN {X 0,Y 261.111,Z 399.275,A -85,B 0,C 180,E1 -18088.458,E2 -18088.458} C_VEL
LIN {X 0,Y 261.13,Z 398.892,A -85,B 0,C 180,E1 -18090,E2 -18090} C_VEL
LIN {X 0,Y 261.125,Z 398.076,A -85,B 0,C 180,E1 -18091.542,E2 -18091.542} C_VEL
LIN {X 0,Y 261.107,Z 396.841,A -85,B 0,C 180,E1 -18093.086,E2 -18093.086} C_VEL
LIN {X 0,Y 261.129,Z 394.445,A -85,B 0,C 180,E1 -18095.23,E2 -18095.23} C_VEL
LIN {X 0,Y 261.357,Z 390.53,A -85,B 0,C 180,E1 -18097.727,E2 -18097.727} C_VEL
LIN {X 0,Y 261.825,Z 385.722,A -85,B 0,C 180,E1 -18100.048,E2 -18100.048} C_VEL
LIN {X 0,Y 262.522,Z 379.628,A -85,B 0,C 180,E1 -18102.367,E2 -18102.367} C_VEL
LIN {X 0,Y 263.742,Z 372.046,A -85,B 0,C 180,E1 -18104.664,E2 -18104.664} C_VEL
LIN {X 0,Y 264.964,Z 364.287,A -85,B 0,C 180,E1 -18106.567,E2 -18106.567} C_VEL
LIN {X 0,Y 266.042,Z 356.34,A -85,B 0,C 180,E1 -18108.183,E2 -18108.183} C_VEL
LIN {X 0,Y 267.38,Z 346.819,A -85,B 0,C 180,E1 -18109.78,E2 -18109.78} C_VEL
LIN {X 0,Y 268.387,Z 338.688,A -85,B 0,C 180,E1 -18110.902,E2 -18110.902} C_VEL
LIN {X 0,Y 267.62,Z 327.898,A -85,B 0,C 180,E1 -18112.251,E2 -18112.251} C_VEL
LIN {X 0,Y 266.455,Z 316.549,A -85,B 0,C 180,E1 -18113.408,E2 -18113.408} C_VEL
LIN {X 0,Y 264.564,Z 303.784,A -85,B 0,C 180,E1 -18114.435,E2 -18114.435} C_VEL
LIN {X 0,Y 262.437,Z 292.917,A -85,B 0,C 180,E1 -18115.153,E2 -18115.153} C_VEL
LIN {X 0,Y 263.164,Z 287.328,A -85,B 0,C 180,E1 -18119.607,E2 -18119.607} C_VEL
LIN {X 0,Y 263.905,Z 283.033,A -85,B 0,C 180,E1 -18123.087,E2 -18123.087} C_VEL
LIN {X 0,Y 264.419,Z 279.789,A -85,B 0,C 180,E1 -18125.784,E2 -18125.784} C_VEL
LIN {X 0,Y 264.383,Z 277.604,A -85,B 0,C 180,E1 -18127.69,E2 -18127.69} C_VEL
LIN {X 0,Y 263.615,Z 273.139,A -85,B 0,C 180,E1 -18131.796,E2 -18131.796} C_VEL
LIN {X 0,Y 263.143,Z 270.709,A -85,B 0,C 180,E1 -18134.282,E2 -18134.282} C_VEL
LIN {X 0,Y 263.077,Z 270.719,A -85,B 0,C 180,E1 -18138.417,E2 -18138.417} C_VEL
LIN {X 0,Y 263.12,Z 270.711,A -85,B 0,C 180,E1 -18142.094,E2 -18142.094} C_VEL
LIN {X 0,Y 263.151,Z 270.704,A -85,B 0,C 180,E1 -18145.884,E2 -18145.884} C_VEL
LIN {X 0,Y 263.122,Z 270.706,A -85,B 0,C 180,E1 -18149.501,E2 -18149.501} C_VEL
LIN {X 0,Y 263.14,Z 270.707,A -85,B 0,C 180,E1 -18152.995,E2 -18152.995} C_VEL
LIN {X 0,Y 263.143,Z 270.706,A -85,B 0,C 180,E1 -18156.381,E2 -18156.381} C_VEL
LIN {X 0,Y 263.246,Z 270.693,A -85,B 0,C 180,E1 -18159.69,E2 -18159.69} C_VEL
LIN {X 0,Y 263.341,Z 270.683,A -85,B 0,C 180,E1 -18164.52,E2 -18164.52} C_VEL
LIN {X 0,Y 263.351,Z 270.676,A -85,B 0,C 180,E1 -18169.232,E2 -18169.232} C_VEL
LIN {X 0,Y 263.554,Z 270.657,A -85,B 0,C 180,E1 -18172.336,E2 -18172.336} C_VEL
LIN {X 0,Y 263.746,Z 270.616,A -85,B 0,C 180,E1 -18178.471,E2 -18178.471} C_VEL
LIN {X 0,Y 263.746,Z 270.622,A -85,B 0,C 180,E1 -18181.525,E2 -18181.525} C_VEL
LIN {X 0,Y 263.566,Z 270.655,A -85,B 0,C 180,E1 -18187.66,E2 -18187.66} C_VEL
LIN {X 0,Y 263.367,Z 270.674,A -85,B 0,C 180,E1 -18190.764,E2 -18190.764} C_VEL
LIN {X 0,Y 263.337,Z 270.682,A -85,B 0,C 180,E1 -18195.477,E2 -18195.477} C_VEL
LIN {X 0,Y 263.256,Z 270.69,A -85,B 0,C 180,E1 -18200.305,E2 -18200.305} C_VEL
LIN {X 0,Y 263.2,Z 270.699,A -85,B 0,C 180,E1 -18205.29,E2 -18205.29} C_VEL
LIN {X 0,Y 263.171,Z 270.701,A -85,B 0,C 180,E1 -18208.728,E2 -18208.728} C_VEL
LIN {X 0,Y 263.124,Z 270.705,A -85,B 0,C 180,E1 -18212.287,E2 -18212.287} C_VEL
LIN {X 0,Y 263.179,Z 270.697,A -85,B 0,C 180,E1 -18215.977,E2 -18215.977} C_VEL
LIN {X 0,Y 263.152,Z 270.703,A -85,B 0,C 180,E1 -18219.861,E2 -18219.861} C_VEL
LIN {X 0,Y 263.196,Z 270.695,A -85,B 0,C 180,E1 -18221.876,E2 -18221.876} C_VEL
LIN {X 0,Y 263.128,Z 270.707,A -85,B 0,C 180,E1 -18226.147,E2 -18226.147} C_VEL
LIN {X 0,Y 263.097,Z 270.711,A -85,B 0,C 180,E1 -18230.127,E2 -18230.127} C_VEL
LIN {X 0,Y 263.176,Z 270.7,A -85,B 0,C 180,E1 -18234.021,E2 -18234.021} C_VEL
LIN {X 0,Y 263.123,Z 270.708,A -85,B 0,C 180,E1 -18237.711,E2 -18237.711} C_VEL
LIN {X 0,Y 263.168,Z 270.702,A -85,B 0,C 180,E1 -18241.792,E2 -18241.792} C_VEL
LIN {X 0,Y 263.109,Z 270.711,A -85,B 0,C 180,E1 -18245.25,E2 -18245.25} C_VEL
LIN {X 0,Y 263.17,Z 270.887,A -85,B 0,C 180,E1 -18247.839,E2 -18247.839} C_VEL
LIN {X 0,Y 262.77,Z 273.966,A -85,B 0,C 180,E1 -18251.28,E2 -18251.28} C_VEL
LIN {X 0,Y 262.615,Z 276.865,A -85,B 0,C 180,E1 -18254.478,E2 -18254.478} C_VEL
LIN {X 0,Y 262.297,Z 280.282,A -85,B 0,C 180,E1 -18257.979,E2 -18257.979} C_VEL
LIN {X 0,Y 265.657,Z 293.537,A -85,B 0,C 180,E1 -18258.943,E2 -18258.943} C_VEL
LIN {X 0,Y 267.689,Z 303.336,A -85,B 0,C 180,E1 -18259.828,E2 -18259.828} C_VEL
LIN {X 0,Y 269.441,Z 315.794,A -85,B 0,C 180,E1 -18261.185,E2 -18261.185} C_VEL
LIN {X 0,Y 269.626,Z 320.506,A -85,B 0,C 180,E1 -18261.758,E2 -18261.758} C_VEL
LIN {X 0,Y 268.046,Z 331.708,A -85,B 0,C 180,E1 -18263.224,E2 -18263.224} C_VEL
LIN {X 0,Y 266.764,Z 340.743,A -85,B 0,C 180,E1 -18264.709,E2 -18264.709} C_VEL
LIN {X 0,Y 265.365,Z 350.022,A -85,B 0,C 180,E1 -18266.584,E2 -18266.584} C_VEL
LIN {X 0,Y 263.979,Z 359.018,A -85,B 0,C 180,E1 -18268.856,E2 -18268.856} C_VEL
LIN {X 0,Y 262.827,Z 366.282,A -85,B 0,C 180,E1 -18271.149,E2 -18271.149} C_VEL
LIN {X 0,Y 262.162,Z 371.182,A -85,B 0,C 180,E1 -18273.073,E2 -18273.073} C_VEL
LIN {X 0,Y 261.673,Z 375.941,A -85,B 0,C 180,E1 -18275.394,E2 -18275.394} C_VEL
LIN {X 0,Y 261.241,Z 379.603,A -85,B 0,C 180,E1 -18277.73,E2 -18277.73} C_VEL
LIN {X 0,Y 261.014,Z 381.497,A -85,B 0,C 180,E1 -18279.297,E2 -18279.297} C_VEL
LIN {X 0,Y 260.863,Z 382.914,A -85,B 0,C 180,E1 -18280.87,E2 -18280.87} C_VEL
LIN {X 0,Y 260.868,Z 383.922,A -85,B 0,C 180,E1 -18282.446,E2 -18282.446} C_VEL
LIN {X 0,Y 260.909,Z 384.574,A -85,B 0,C 180,E1 -18284.146,E2 -18284.146} C_VEL
LIN {X 0,Y 260.943,Z 384.733,A -85,B 0,C 180,E1 -18285.624,E2 -18285.624} C_VEL
LIN {X 0,Y 261.123,Z 384.487,A -85,B 0,C 180,E1 -18287.221,E2 -18287.221} C_VEL
LIN {X 0,Y 261.741,Z 383.09,A -85,B 0,C 180,E1 -18289.992,E2 -18289.992} C_VEL
LIN {X 0,Y 262.405,Z 381.245,A -85,B 0,C 180,E1 -18292.021,E2 -18292.021} C_VEL
LIN {X 0,Y 263.766,Z 377.083,A -85,B 0,C 180,E1 -18295.058,E2 -18295.058} C_VEL
LIN {X 0,Y 265.397,Z 372.113,A -85,B 0,C 180,E1 -18297.607,E2 -18297.607} C_VEL
LIN {X 0,Y 267.323,Z 366.063,A -85,B 0,C 180,E1 -18299.967,E2 -18299.967} C_VEL
LIN {X 0,Y 269.616,Z 358.446,A -85,B 0,C 180,E1 -18302.3,E2 -18302.3} C_VEL
LIN {X 0,Y 271.921,Z 350.364,A -85,B 0,C 180,E1 -18304.27,E2 -18304.27} C_VEL
LIN {X 0,Y 274.337,Z 341.015,A -85,B 0,C 180,E1 -18306.1,E2 -18306.1} C_VEL
LIN {X 0,Y 276.909,Z 329.769,A -85,B 0,C 180,E1 -18307.83,E2 -18307.83} C_VEL
LIN {X 0,Y 276.61,Z 324.857,A -85,B 0,C 180,E1 -18308.626,E2 -18308.626} C_VEL
LIN {X 0,Y 274.661,Z 313.849,A -85,B 0,C 180,E1 -18310.341,E2 -18310.341} C_VEL
LIN {X 0,Y 272.054,Z 303.845,A -85,B 0,C 180,E1 -18311.764,E2 -18311.764} C_VEL
LIN {X 0,Y 267.974,Z 291.957,A -85,B 0,C 180,E1 -18313.344,E2 -18313.344} C_VEL
LIN {X 0,Y 264.384,Z 283.841,A -85,B 0,C 180,E1 -18314.39,E2 -18314.39} C_VEL
LIN {X 0,Y 263.481,Z 280.907,A -85,B 0,C 180,E1 -18314.703,E2 -18314.703} C_VEL
LIN {X 0,Y 263.827,Z 278.137,A -85,B 0,C 180,E1 -18318.246,E2 -18318.246} C_VEL
LIN {X 0,Y 263.829,Z 276.435,A -85,B 0,C 180,E1 -18320.579,E2 -18320.579} C_VEL
LIN {X 0,Y 263.608,Z 274.025,A -85,B 0,C 180,E1 -18324.091,E2 -18324.091} C_VEL
LIN {X 0,Y 263.304,Z 271.716,A -85,B 0,C 180,E1 -18327.738,E2 -18327.738} C_VEL
LIN {X 0,Y 263.14,Z 270.709,A -85,B 0,C 180,E1 -18329.508,E2 -18329.508} C_VEL
LIN {X 0,Y 263.185,Z 270.7,A -85,B 0,C 180,E1 -18333.004,E2 -18333.004} C_VEL
LIN {X 0,Y 263.185,Z 270.701,A -85,B 0,C 180,E1 -18336.389,E2 -18336.389} C_VEL
LIN {X 0,Y 263.28,Z 270.686,A -85,B 0,C 180,E1 -18339.697,E2 -18339.697} C_VEL
LIN {X 0,Y 263.337,Z 270.682,A -85,B 0,C 180,E1 -18344.523,E2 -18344.523} C_VEL
LIN {X 0,Y 263.347,Z 270.682,A -85,B 0,C 180,E1 -18349.235,E2 -18349.235} C_VEL
LIN {X 0,Y 263.55,Z 270.656,A -85,B 0,C 180,E1 -18352.34,E2 -18352.34} C_VEL
LIN {X 0,Y 263.745,Z 270.633,A -85,B 0,C 180,E1 -18358.475,E2 -18358.475} C_VEL
LIN {X 0,Y 263.744,Z 270.631,A -85,B 0,C 180,E1 -18361.529,E2 -18361.529} C_VEL
LIN {X 0,Y 263.567,Z 270.654,A -85,B 0,C 180,E1 -18367.664,E2 -18367.664} C_VEL
LIN {X 0,Y 263.369,Z 270.68,A -85,B 0,C 180,E1 -18370.768,E2 -18370.768} C_VEL
LIN {X 0,Y 263.341,Z 270.684,A -85,B 0,C 180,E1 -18375.48,E2 -18375.48} C_VEL
LIN {X 0,Y 263.261,Z 270.698,A -85,B 0,C 180,E1 -18380.309,E2 -18380.309} C_VEL
LIN {X 0,Y 263.14,Z 270.714,A -85,B 0,C 180,E1 -18383.447,E2 -18383.447} C_VEL
LIN {X 0,Y 262.522,Z 270.797,A -85,B 0,C 180,E1 -18384.726,E2 -18384.726} C_VEL
LIN {X 0,Y 259.659,Z 271.154,A -85,B 0,C 180,E1 -18386.808,E2 -18386.808} C_VEL
LIN {X 0,Y 257.191,Z 271.456,A -85,B 0,C 180,E1 -18388.503,E2 -18388.503} C_VEL
LIN {X 0,Y 256.126,Z 271.586,A -85,B 0,C 180,E1 -18389.818,E2 -18389.818} C_VEL
LIN {X 0,Y 256.039,Z 271.593,A -85,B 0,C 180,E1 -18390.264,E2 -18390.264} C_VEL
LIN {X 0,Y 256.065,Z 271.59,A -85,B 0,C 180,E1 -18393.295,E2 -18393.295} C_VEL
LIN {X 0,Y 256.608,Z 274.15,A -85,B 0,C 180,E1 -18397.417,E2 -18397.417} C_VEL
LIN {X 0,Y 256.989,Z 276.8,A -85,B 0,C 180,E1 -18401.023,E2 -18401.023} C_VEL
LIN {X 0,Y 257.488,Z 280.195,A -85,B 0,C 180,E1 -18405.209,E2 -18405.209} C_VEL
LIN {X 0,Y 258.055,Z 283.676,A -85,B 0,C 180,E1 -18409.186,E2 -18409.186} C_VEL
LIN {X 0,Y 258.294,Z 286.454,A -85,B 0,C 180,E1 -18412.101,E2 -18412.101} C_VEL
LIN {X 0,Y 258.079,Z 289.55,A -85,B 0,C 180,E1 -18415.12,E2 -18415.12} C_VEL
LIN {X 0,Y 257.532,Z 292.026,A -85,B 0,C 180,E1 -18417.365,E2 -18417.365} C_VEL
LIN {X 0,Y 258.562,Z 295.387,A -85,B 0,C 180,E1 -18417.703,E2 -18417.703} C_VEL
LIN {X 0,Y 261.99,Z 305.139,A -85,B 0,C 180,E1 -18418.861,E2 -18418.861} C_VEL
LIN {X 0,Y 265.068,Z 316.438,A -85,B 0,C 180,E1 -18420.287,E2 -18420.287} C_VEL
LIN {X 0,Y 267.152,Z 327.026,A -85,B 0,C 180,E1 -18421.737,E2 -18421.737} C_VEL
LIN {X 0,Y 268.309,Z 337.437,A -85,B 0,C 180,E1 -18423.291,E2 -18423.291} C_VEL
LIN {X 0,Y 268.616,Z 346.783,A -85,B 0,C 180,E1 -18424.84,E2 -18424.84} C_VEL
LIN {X 0,Y 267.462,Z 352.409,A -85,B 0,C 180,E1 -18425.76,E2 -18425.76} C_VEL
LIN {X 0,Y 264.984,Z 361.184,A -85,B 0,C 180,E1 -18427.383,E2 -18427.383} C_VEL
LIN {X 0,Y 262.626,Z 369.265,A -85,B 0,C 180,E1 -18429.233,E2 -18429.233} C_VEL
LIN {X 0,Y 260.336,Z 377.214,A -85,B 0,C 180,E1 -18431.507,E2 -18431.507} C_VEL
LIN {X 0,Y 258.648,Z 382.624,A -85,B 0,C 180,E1 -18433.423,E2 -18433.423} C_VEL
LIN {X 0,Y 256.826,Z 387.946,A -85,B 0,C 180,E1 -18435.743,E2 -18435.743} C_VEL
LIN {X 0,Y 255.633,Z 392.115,A -85,B 0,C 180,E1 -18438.101,E2 -18438.101} C_VEL
LIN {X 0,Y 254.776,Z 395.252,A -85,B 0,C 180,E1 -18440.473,E2 -18440.473} C_VEL
LIN {X 0,Y 254.362,Z 396.828,A -85,B 0,C 180,E1 -18442.059,E2 -18442.059} C_VEL
LIN {X 0,Y 253.988,Z 398.644,A -85,B 0,C 180,E1 -18444.979,E2 -18444.979} C_VEL
LIN {X 0,Y 253.957,Z 399.085,A -85,B 0,C 180,E1 -18446.827,E2 -18446.827} C_VEL
LIN {X 0,Y 254.017,Z 399.062,A -85,B 0,C 180,E1 -18448.415,E2 -18448.415} C_VEL
LIN {X 0,Y 254.058,Z 398.644,A -85,B 0,C 180,E1 -18450,E2 -18450} C_VEL
LIN {X 0,Y 254.054,Z 397.787,A -85,B 0,C 180,E1 -18451.585,E2 -18451.585} C_VEL
LIN {X 0,Y 254.003,Z 396.525,A -85,B 0,C 180,E1 -18453.172,E2 -18453.172} C_VEL
LIN {X 0,Y 254.027,Z 394.422,A -85,B 0,C 180,E1 -18455.119,E2 -18455.119} C_VEL
LIN {X 0,Y 254.313,Z 390.102,A -85,B 0,C 180,E1 -18457.942,E2 -18457.942} C_VEL
LIN {X 0,Y 254.79,Z 385.231,A -85,B 0,C 180,E1 -18460.328,E2 -18460.328} C_VEL
LIN {X 0,Y 255.55,Z 379.069,A -85,B 0,C 180,E1 -18462.71,E2 -18462.71} C_VEL
LIN {X 0,Y 256.834,Z 371.408,A -85,B 0,C 180,E1 -18465.067,E2 -18465.067} C_VEL
LIN {X 0,Y 258.096,Z 363.543,A -85,B 0,C 180,E1 -18467.021,E2 -18467.021} C_VEL
LIN {X 0,Y 259.194,Z 355.786,A -85,B 0,C 180,E1 -18468.624,E2 -18468.624} C_VEL
LIN {X 0,Y 260.671,Z 345.81,A -85,B 0,C 180,E1 -18470.311,E2 -18470.311} C_VEL
LIN {X 0,Y 261.445,Z 339,A -85,B 0,C 180,E1 -18471.278,E2 -18471.278} C_VEL
LIN {X 0,Y 260.624,Z 326.973,A -85,B 0,C 180,E1 -18472.823,E2 -18472.823} C_VEL
LIN {X 0,Y 259.284,Z 314.474,A -85,B 0,C 180,E1 -18474.096,E2 -18474.096} C_VEL
LIN {X 0,Y 257.301,Z 301.912,A -85,B 0,C 180,E1 -18475.11,E2 -18475.11} C_VEL
LIN {X 0,Y 255.452,Z 292.741,A -85,B 0,C 180,E1 -18475.727,E2 -18475.727} C_VEL
LIN {X 0,Y 256.264,Z 286.951,A -85,B 0,C 180,E1 -18480.487,E2 -18480.487} C_VEL
LIN {X 0,Y 257.071,Z 282.691,A -85,B 0,C 180,E1 -18484.055,E2 -18484.055} C_VEL
LIN {X 0,Y 257.376,Z 279.399,A -85,B 0,C 180,E1 -18486.922,E2 -18486.922} C_VEL
LIN {X 0,Y 256.746,Z 274.967,A -85,B 0,C 180,E1 -18491.067,E2 -18491.067} C_VEL
LIN {X 0,Y 256.099,Z 271.587,A -85,B 0,C 180,E1 -18494.477,E2 -18494.477} C_VEL
LIN {X 0,Y 256.016,Z 271.601,A -85,B 0,C 180,E1 -18498.787,E2 -18498.787} C_VEL
LIN {X 0,Y 256.099,Z 271.587,A -85,B 0,C 180,E1 -18502.86,E2 -18502.86} C_VEL
LIN {X 0,Y 256.066,Z 271.591,A -85,B 0,C 180,E1 -18506.705,E2 -18506.705} C_VEL
LIN {X 0,Y 256.051,Z 271.589,A -85,B 0,C 180,E1 -18510.391,E2 -18510.391} C_VEL
LIN {X 0,Y 256.131,Z 271.578,A -85,B 0,C 180,E1 -18514.887,E2 -18514.887} C_VEL
LIN {X 0,Y 256.145,Z 271.577,A -85,B 0,C 180,E1 -18519.101,E2 -18519.101} C_VEL
LIN {X 0,Y 256.258,Z 271.562,A -85,B 0,C 180,E1 -18523.713,E2 -18523.713} C_VEL
LIN {X 0,Y 256.29,Z 271.558,A -85,B 0,C 180,E1 -18527.326,E2 -18527.326} C_VEL
LIN {X 0,Y 256.511,Z 271.536,A -85,B 0,C 180,E1 -18532.124,E2 -18532.124} C_VEL
LIN {X 0,Y 256.492,Z 271.526,A -85,B 0,C 180,E1 -18536.857,E2 -18536.857} C_VEL
LIN {X 0,Y 256.768,Z 271.486,A -85,B 0,C 180,E1 -18539.998,E2 -18539.998} C_VEL
LIN {X 0,Y 256.494,Z 271.529,A -85,B 0,C 180,E1 -18543.139,E2 -18543.139} C_VEL
LIN {X 0,Y 256.533,Z 271.529,A -85,B 0,C 180,E1 -18547.871,E2 -18547.871} C_VEL
LIN {X 0,Y 256.303,Z 271.555,A -85,B 0,C 180,E1 -18551.064,E2 -18551.064} C_VEL
LIN {X 0,Y 256.272,Z 271.558,A -85,B 0,C 180,E1 -18555.915,E2 -18555.915} C_VEL
LIN {X 0,Y 256.159,Z 271.576,A -85,B 0,C 180,E1 -18560.894,E2 -18560.894} C_VEL
LIN {X 0,Y 256.18,Z 271.571,A -85,B 0,C 180,E1 -18565.137,E2 -18565.137} C_VEL
LIN {X 0,Y 256.105,Z 271.578,A -85,B 0,C 180,E1 -18569.598,E2 -18569.598} C_VEL
LIN {X 0,Y 256.076,Z 271.587,A -85,B 0,C 180,E1 -18573.289,E2 -18573.289} C_VEL
LIN {X 0,Y 256.131,Z 271.579,A -85,B 0,C 180,E1 -18577.277,E2 -18577.277} C_VEL
LIN {X 0,Y 256.121,Z 271.579,A -85,B 0,C 180,E1 -18581.187,E2 -18581.187} C_VEL
LIN {X 0,Y 256.062,Z 271.587,A -85,B 0,C 180,E1 -18585.526,E2 -18585.526} C_VEL
LIN {X 0,Y 256.049,Z 271.59,A -85,B 0,C 180,E1 -18588.797,E2 -18588.797} C_VEL
LIN {X 0,Y 256.133,Z 271.579,A -85,B 0,C 180,E1 -18592.869,E2 -18592.869} C_VEL
LIN {X 0,Y 256.075,Z 271.589,A -85,B 0,C 180,E1 -18596.709,E2 -18596.709} C_VEL
LIN {X 0,Y 256.088,Z 271.587,A -85,B 0,C 180,E1 -18600.398,E2 -18600.398} C_VEL
LIN {X 0,Y 256.083,Z 271.586,A -85,B 0,C 180,E1 -18603.954,E2 -18603.954} C_VEL
LIN {X 0,Y 256.098,Z 271.653,A -85,B 0,C 180,E1 -18607.62,E2 -18607.62} C_VEL
LIN {X 0,Y 255.766,Z 274.409,A -85,B 0,C 180,E1 -18610.748,E2 -18610.748} C_VEL
LIN {X 0,Y 255.563,Z 277.488,A -85,B 0,C 180,E1 -18614.251,E2 -18614.251} C_VEL
LIN {X 0,Y 255.24,Z 280.338,A -85,B 0,C 180,E1 -18617.369,E2 -18617.369} C_VEL
LIN {X 0,Y 258.893,Z 294.672,A -85,B 0,C 180,E1 -18618.479,E2 -18618.479} C_VEL
LIN {X 0,Y 261.129,Z 306.009,A -85,B 0,C 180,E1 -18619.57,E2 -18619.57} C_VEL
LIN {X 0,Y 262.731,Z 317.978,A -85,B 0,C 180,E1 -18620.958,E2 -18620.958} C_VEL
LIN {X 0,Y 262.618,Z 322.584,A -85,B 0,C 180,E1 -18621.536,E2 -18621.536} C_VEL
LIN {X 0,Y 261.017,Z 333.352,A -85,B 0,C 180,E1 -18623.041,E2 -18623.041} C_VEL
LIN {X 0,Y 259.728,Z 342.138,A -85,B 0,C 180,E1 -18624.566,E2 -18624.566} C_VEL
LIN {X 0,Y 258.249,Z 351.2,A -85,B 0,C 180,E1 -18626.49,E2 -18626.49} C_VEL
LIN {X 0,Y 256.834,Z 360.034,A -85,B 0,C 180,E1 -18628.824,E2 -18628.824} C_VEL
LIN {X 0,Y 255.734,Z 367.119,A -85,B 0,C 180,E1 -18631.181,E2 -18631.181} C_VEL
LIN {X 0,Y 254.852,Z 373.582,A -85,B 0,C 180,E1 -18633.953,E2 -18633.953} C_VEL
LIN {X 0,Y 254.411,Z 377.85,A -85,B 0,C 180,E1 -18636.344,E2 -18636.344} C_VEL
LIN {X 0,Y 254.103,Z 380.129,A -85,B 0,C 180,E1 -18637.949,E2 -18637.949} C_VEL
LIN {X 0,Y 253.876,Z 381.927,A -85,B 0,C 180,E1 -18639.561,E2 -18639.561} C_VEL
LIN {X 0,Y 253.759,Z 383.288,A -85,B 0,C 180,E1 -18641.178,E2 -18641.178} C_VEL
LIN {X 0,Y 253.835,Z 384.775,A -85,B 0,C 180,E1 -18644.301,E2 -18644.301} C_VEL
LIN {X 0,Y 253.884,Z 384.913,A -85,B 0,C 180,E1 -18646.07,E2 -18646.07} C_VEL
LIN {X 0,Y 254.101,Z 384.618,A -85,B 0,C 180,E1 -18647.712,E2 -18647.712} C_VEL
LIN {X 0,Y 254.736,Z 383.313,A -85,B 0,C 180,E1 -18650.283,E2 -18650.283} C_VEL
LIN {X 0,Y 255.885,Z 380.227,A -85,B 0,C 180,E1 -18653.468,E2 -18653.468} C_VEL
LIN {X 0,Y 257.165,Z 376.595,A -85,B 0,C 180,E1 -18655.928,E2 -18655.928} C_VEL
LIN {X 0,Y 258.826,Z 371.766,A -85,B 0,C 180,E1 -18658.371,E2 -18658.371} C_VEL
LIN {X 0,Y 260.863,Z 365.583,A -85,B 0,C 180,E1 -18660.789,E2 -18660.789} C_VEL
LIN {X 0,Y 263.336,Z 357.82,A -85,B 0,C 180,E1 -18663.168,E2 -18663.168} C_VEL
LIN {X 0,Y 265.927,Z 349.041,A -85,B 0,C 180,E1 -18665.279,E2 -18665.279} C_VEL
LIN {X 0,Y 268.68,Z 338.808,A -85,B 0,C 180,E1 -18667.22,E2 -18667.22} C_VEL
LIN {X 0,Y 270.543,Z 330.144,A -85,B 0,C 180,E1 -18668.568,E2 -18668.568} C_VEL
LIN {X 0,Y 269.266,Z 320.344,A -85,B 0,C 180,E1 -18670.235,E2 -18670.235} C_VEL
LIN {X 0,Y 267.115,Z 310.162,A -85,B 0,C 180,E1 -18671.822,E2 -18671.822} C_VEL
LIN {X 0,Y 263.754,Z 299.063,A -85,B 0,C 180,E1 -18673.442,E2 -18673.442} C_VEL
LIN {X 0,Y 259.669,Z 288.669,A -85,B 0,C 180,E1 -18674.886,E2 -18674.886} C_VEL
LIN {X 0,Y 256.707,Z 281.824,A -85,B 0,C 180,E1 -18675.784,E2 -18675.784} C_VEL
LIN {X 0,Y 256.602,Z 281.13,A -85,B 0,C 180,E1 -18675.876,E2 -18675.876} C_VEL
LIN {X 0,Y 256.804,Z 278.831,A -85,B 0,C 180,E1 -18678.946,E2 -18678.946} C_VEL
LIN {X 0,Y 256.732,Z 276.337,A -85,B 0,C 180,E1 -18682.547,E2 -18682.547} C_VEL
LIN {X 0,Y 256.392,Z 273.677,A -85,B 0,C 180,E1 -18686.757,E2 -18686.757} C_VEL
LIN {X 0,Y 256.102,Z 271.587,A -85,B 0,C 180,E1 -18690.401,E2 -18690.401} C_VEL
LIN {X 0,Y 256.182,Z 271.572,A -85,B 0,C 180,E1 -18694.862,E2 -18694.862} C_VEL
LIN {X 0,Y 256.228,Z 271.565,A -85,B 0,C 180,E1 -18699.112,E2 -18699.112} C_VEL
LIN {X 0,Y 256.287,Z 271.562,A -85,B 0,C 180,E1 -18704.086,E2 -18704.086} C_VEL
LIN {X 0,Y 256.289,Z 271.562,A -85,B 0,C 180,E1 -18708.935,E2 -18708.935} C_VEL
LIN {X 0,Y 256.508,Z 271.534,A -85,B 0,C 180,E1 -18712.128,E2 -18712.128} C_VEL
LIN {X 0,Y 256.492,Z 271.536,A -85,B 0,C 180,E1 -18716.86,E2 -18716.86} C_VEL
LIN {X 0,Y 256.751,Z 271.502,A -85,B 0,C 180,E1 -18720.002,E2 -18720.002} C_VEL
LIN {X 0,Y 256.493,Z 271.536,A -85,B 0,C 180,E1 -18723.143,E2 -18723.143} C_VEL
LIN {X 0,Y 256.535,Z 271.529,A -85,B 0,C 180,E1 -18727.875,E2 -18727.875} C_VEL
LIN {X 0,Y 256.305,Z 271.56,A -85,B 0,C 180,E1 -18731.068,E2 -18731.068} C_VEL
LIN {X 0,Y 256.291,Z 271.564,A -85,B 0,C 180,E1 -18735.917,E2 -18735.917} C_VEL
LIN {X 0,Y 256.162,Z 271.581,A -85,B 0,C 180,E1 -18740.897,E2 -18740.897} C_VEL
LIN {X 0,Y 256.164,Z 271.585,A -85,B 0,C 180,E1 -18745.13,E2 -18745.13} C_VEL
LIN {X 0,Y 256.11,Z 271.59,A -85,B 0,C 180,E1 -18748.586,E2 -18748.586} C_VEL
LIN {X 0,Y 256.039,Z 271.593,A -85,B 0,C 180,E1 -18750.264,E2 -18750.264} C_VEL
LIN {X 0,Y 255.397,Z 271.828,A -85,B 0,C 180,E1 -18751.577,E2 -18751.577} C_VEL
LIN {X 0,Y 252.697,Z 272.98,A -85,B 0,C 180,E1 -18753.713,E2 -18753.713} C_VEL
LIN {X 0,Y 250.474,Z 274.265,A -85,B 0,C 180,E1 -18755.445,E2 -18755.445} C_VEL
LIN {X 0,Y 249.617,Z 275.255,A -85,B 0,C 180,E1 -18756.781,E2 -18756.781} C_VEL
LIN {X 0,Y 249.598,Z 275.565,A -85,B 0,C 180,E1 -18757.233,E2 -18757.233} C_VEL
LIN {X 0,Y 250.004,Z 277.963,A -85,B 0,C 180,E1 -18760.625,E2 -18760.625} C_VEL
LIN {X 0,Y 250.443,Z 281.005,A -85,B 0,C 180,E1 -18764.554,E2 -18764.554} C_VEL
LIN {X 0,Y 251.066,Z 284.875,A -85,B 0,C 180,E1 -18769.098,E2 -18769.098} C_VEL
LIN {X 0,Y 251.317,Z 287.582,A -85,B 0,C 180,E1 -18772.033,E2 -18772.033} C_VEL
LIN {X 0,Y 251.137,Z 289.788,A -85,B 0,C 180,E1 -18774.251,E2 -18774.251} C_VEL
LIN {X 0,Y 250.764,Z 291.753,A -85,B 0,C 180,E1 -18776.146,E2 -18776.146} C_VEL
LIN {X 0,Y 251.774,Z 295.092,A -85,B 0,C 180,E1 -18776.512,E2 -18776.512} C_VEL
LIN {X 0,Y 255.428,Z 305.252,A -85,B 0,C 180,E1 -18777.81,E2 -18777.81} C_VEL
LIN {X 0,Y 258.502,Z 316.4,A -85,B 0,C 180,E1 -18779.296,E2 -18779.296} C_VEL
LIN {X 0,Y 260.776,Z 328.068,A -85,B 0,C 180,E1 -18780.981,E2 -18780.981} C_VEL
LIN {X 0,Y 261.879,Z 338.463,A -85,B 0,C 180,E1 -18782.621,E2 -18782.621} C_VEL
LIN {X 0,Y 262.071,Z 348.535,A -85,B 0,C 180,E1 -18784.384,E2 -18784.384} C_VEL
LIN {X 0,Y 259.586,Z 357.929,A -85,B 0,C 180,E1 -18786.04,E2 -18786.04} C_VEL
LIN {X 0,Y 256.926,Z 366.562,A -85,B 0,C 180,E1 -18787.907,E2 -18787.907} C_VEL
LIN {X 0,Y 254.466,Z 374.552,A -85,B 0,C 180,E1 -18790.081,E2 -18790.081} C_VEL
LIN {X 0,Y 252.22,Z 381.751,A -85,B 0,C 180,E1 -18792.57,E2 -18792.57} C_VEL
LIN {X 0,Y 249.942,Z 388.012,A -85,B 0,C 180,E1 -18795.341,E2 -18795.341} C_VEL
LIN {X 0,Y 248.664,Z 392.12,A -85,B 0,C 180,E1 -18797.762,E2 -18797.762} C_VEL
LIN {X 0,Y 247.742,Z 395.199,A -85,B 0,C 180,E1 -18800.2,E2 -18800.2} C_VEL
LIN {X 0,Y 247.31,Z 396.745,A -85,B 0,C 180,E1 -18801.832,E2 -18801.832} C_VEL
LIN {X 0,Y 246.888,Z 398.564,A -85,B 0,C 180,E1 -18805.101,E2 -18805.101} C_VEL
LIN {X 0,Y 246.925,Z 398.849,A -85,B 0,C 180,E1 -18808.369,E2 -18808.369} C_VEL
LIN {X 0,Y 246.987,Z 398.384,A -85,B 0,C 180,E1 -18810,E2 -18810} C_VEL
LIN {X 0,Y 246.961,Z 397.497,A -85,B 0,C 180,E1 -18811.631,E2 -18811.631} C_VEL
LIN {X 0,Y 246.905,Z 396.208,A -85,B 0,C 180,E1 -18813.264,E2 -18813.264} C_VEL
LIN {X 0,Y 246.956,Z 394.292,A -85,B 0,C 180,E1 -18815.081,E2 -18815.081} C_VEL
LIN {X 0,Y 247.124,Z 391.074,A -85,B 0,C 180,E1 -18817.353,E2 -18817.353} C_VEL
LIN {X 0,Y 247.581,Z 386.54,A -85,B 0,C 180,E1 -18819.806,E2 -18819.806} C_VEL
LIN {X 0,Y 248.277,Z 380.761,A -85,B 0,C 180,E1 -18822.257,E2 -18822.257} C_VEL
LIN {X 0,Y 249.455,Z 373.503,A -85,B 0,C 180,E1 -18824.688,E2 -18824.688} C_VEL
LIN {X 0,Y 250.997,Z 364.473,A -85,B 0,C 180,E1 -18827.097,E2 -18827.097} C_VEL
LIN {X 0,Y 251.999,Z 357.529,A -85,B 0,C 180,E1 -18828.622,E2 -18828.622} C_VEL
LIN {X 0,Y 253.577,Z 347.261,A -85,B 0,C 180,E1 -18830.481,E2 -18830.481} C_VEL
LIN {X 0,Y 254.519,Z 339.276,A -85,B 0,C 180,E1 -18831.673,E2 -18831.673} C_VEL
LIN {X 0,Y 253.768,Z 327.493,A -85,B 0,C 180,E1 -18833.245,E2 -18833.245} C_VEL
LIN {X 0,Y 252.572,Z 315.831,A -85,B 0,C 180,E1 -18834.505,E2 -18834.505} C_VEL
LIN {X 0,Y 250.587,Z 303.004,A -85,B 0,C 180,E1 -18835.605,E2 -18835.605} C_VEL
LIN {X 0,Y 248.46,Z 292.521,A -85,B 0,C 180,E1 -18836.376,E2 -18836.376} C_VEL
LIN {X 0,Y 249.413,Z 286.575,A -85,B 0,C 180,E1 -18841.419,E2 -18841.419} C_VEL
LIN {X 0,Y 250.26,Z 281.914,A -85,B 0,C 180,E1 -18845.469,E2 -18845.469} C_VEL
LIN {X 0,Y 250.212,Z 279.002,A -85,B 0,C 180,E1 -18848.165,E2 -18848.165} C_VEL
LIN {X 0,Y 249.424,Z 274.192,A -85,B 0,C 180,E1 -18852.893,E2 -18852.893} C_VEL
LIN {X 0,Y 249.024,Z 272.47,A -85,B 0,C 180,E1 -18854.873,E2 -18854.873} C_VEL
LIN {X 0,Y 248.982,Z 272.473,A -85,B 0,C 180,E1 -18859.651,E2 -18859.651} C_VEL
LIN {X 0,Y 249.011,Z 272.467,A -85,B 0,C 180,E1 -18863.649,E2 -18863.649} C_VEL
LIN {X 0,Y 249.032,Z 272.463,A -85,B 0,C 180,E1 -18867.846,E2 -18867.846} C_VEL
LIN {X 0,Y 249.045,Z 272.46,A -85,B 0,C 180,E1 -18871.33,E2 -18871.33} C_VEL
LIN {X 0,Y 249.1,Z 272.453,A -85,B 0,C 180,E1 -18874.961,E2 -18874.961} C_VEL
LIN {X 0,Y 249.087,Z 272.459,A -85,B 0,C 180,E1 -18878.603,E2 -18878.603} C_VEL
LIN {X 0,Y 249.221,Z 272.438,A -85,B 0,C 180,E1 -18883.619,E2 -18883.619} C_VEL
LIN {X 0,Y 249.241,Z 272.435,A -85,B 0,C 180,E1 -18888.614,E2 -18888.614} C_VEL
LIN {X 0,Y 249.451,Z 272.414,A -85,B 0,C 180,E1 -18891.9,E2 -18891.9} C_VEL
LIN {X 0,Y 249.29,Z 272.428,A -85,B 0,C 180,E1 -18895.146,E2 -18895.146} C_VEL
LIN {X 0,Y 249.671,Z 272.367,A -85,B 0,C 180,E1 -18898.385,E2 -18898.385} C_VEL
LIN {X 0,Y 249.671,Z 272.374,A -85,B 0,C 180,E1 -18901.611,E2 -18901.611} C_VEL
LIN {X 0,Y 249.443,Z 272.41,A -85,B 0,C 180,E1 -18906.777,E2 -18906.777} C_VEL
LIN {X 0,Y 249.383,Z 272.418,A -85,B 0,C 180,E1 -18909.733,E2 -18909.733} C_VEL
LIN {X 0,Y 249.19,Z 272.442,A -85,B 0,C 180,E1 -18914.702,E2 -18914.702} C_VEL
LIN {X 0,Y 249.128,Z 272.45,A -85,B 0,C 180,E1 -18918.076,E2 -18918.076} C_VEL
LIN {X 0,Y 249.08,Z 272.458,A -85,B 0,C 180,E1 -18921.516,E2 -18921.516} C_VEL
LIN {X 0,Y 249.123,Z 272.453,A -85,B 0,C 180,E1 -18925.48,E2 -18925.48} C_VEL
LIN {X 0,Y 249.075,Z 272.458,A -85,B 0,C 180,E1 -18928.992,E2 -18928.992} C_VEL
LIN {X 0,Y 249.027,Z 272.461,A -85,B 0,C 180,E1 -18932.424,E2 -18932.424} C_VEL
LIN {X 0,Y 249.065,Z 272.455,A -85,B 0,C 180,E1 -18936.337,E2 -18936.337} C_VEL
LIN {X 0,Y 249.074,Z 272.458,A -85,B 0,C 180,E1 -18940.462,E2 -18940.462} C_VEL
LIN {X 0,Y 249.064,Z 272.457,A -85,B 0,C 180,E1 -18942.807,E2 -18942.807} C_VEL
LIN {X 0,Y 249.015,Z 272.461,A -85,B 0,C 180,E1 -18947.364,E2 -18947.364} C_VEL
LIN {X 0,Y 249.042,Z 272.462,A -85,B 0,C 180,E1 -18952.197,E2 -18952.197} C_VEL
LIN {X 0,Y 249.051,Z 272.46,A -85,B 0,C 180,E1 -18955.641,E2 -18955.641} C_VEL
LIN {X 0,Y 249.035,Z 272.463,A -85,B 0,C 180,E1 -18959.472,E2 -18959.472} C_VEL
LIN {X 0,Y 249.034,Z 272.463,A -85,B 0,C 180,E1 -18963.158,E2 -18963.158} C_VEL
LIN {X 0,Y 249.086,Z 272.597,A -85,B 0,C 180,E1 -18967.611,E2 -18967.611} C_VEL
LIN {X 0,Y 248.613,Z 276.284,A -85,B 0,C 180,E1 -18971.883,E2 -18971.883} C_VEL
LIN {X 0,Y 248.414,Z 279.201,A -85,B 0,C 180,E1 -18975.249,E2 -18975.249} C_VEL
LIN {X 0,Y 248.241,Z 280.541,A -85,B 0,C 180,E1 -18976.754,E2 -18976.754} C_VEL
LIN {X 0,Y 251.831,Z 294.394,A -85,B 0,C 180,E1 -18977.863,E2 -18977.863} C_VEL
LIN {X 0,Y 253.994,Z 304.887,A -85,B 0,C 180,E1 -18978.897,E2 -18978.897} C_VEL
LIN {X 0,Y 255.704,Z 317.134,A -85,B 0,C 180,E1 -18980.339,E2 -18980.339} C_VEL
LIN {X 0,Y 256.015,Z 321.471,A -85,B 0,C 180,E1 -18980.918,E2 -18980.918} C_VEL
LIN {X 0,Y 254.314,Z 332.568,A -85,B 0,C 180,E1 -18982.457,E2 -18982.457} C_VEL
LIN {X 0,Y 252.945,Z 341.524,A -85,B 0,C 180,E1 -18984.019,E2 -18984.019} C_VEL
LIN {X 0,Y 251.454,Z 350.719,A -85,B 0,C 180,E1 -18985.993,E2 -18985.993} C_VEL
LIN {X 0,Y 249.948,Z 359.671,A -85,B 0,C 180,E1 -18988.389,E2 -18988.389} C_VEL
LIN {X 0,Y 248.74,Z 366.888,A -85,B 0,C 180,E1 -18990.809,E2 -18990.809} C_VEL
LIN {X 0,Y 247.904,Z 372.64,A -85,B 0,C 180,E1 -18993.25,E2 -18993.25} C_VEL
LIN {X 0,Y 247.376,Z 377.787,A -85,B 0,C 180,E1 -18996.113,E2 -18996.113} C_VEL
LIN {X 0,Y 246.965,Z 380.624,A -85,B 0,C 180,E1 -18998.18,E2 -18998.18} C_VEL
LIN {X 0,Y 246.76,Z 382.346,A -85,B 0,C 180,E1 -18999.839,E2 -18999.839} C_VEL
LIN {X 0,Y 246.666,Z 383.659,A -85,B 0,C 180,E1 -19001.504,E2 -19001.504} C_VEL
LIN {X 0,Y 246.721,Z 384.964,A -85,B 0,C 180,E1 -19004.427,E2 -19004.427} C_VEL
LIN {X 0,Y 246.837,Z 385.093,A -85,B 0,C 180,E1 -19006.542,E2 -19006.542} C_VEL
LIN {X 0,Y 247.105,Z 384.75,A -85,B 0,C 180,E1 -19008.231,E2 -19008.231} C_VEL
LIN {X 0,Y 247.721,Z 383.548,A -85,B 0,C 180,E1 -19010.579,E2 -19010.579} C_VEL
LIN {X 0,Y 248.697,Z 381.109,A -85,B 0,C 180,E1 -19013.305,E2 -19013.305} C_VEL
LIN {X 0,Y 250.045,Z 377.605,A -85,B 0,C 180,E1 -19015.923,E2 -19015.923} C_VEL
LIN {X 0,Y 251.655,Z 373.22,A -85,B 0,C 180,E1 -19018.343,E2 -19018.343} C_VEL
LIN {X 0,Y 254.023,Z 366.497,A -85,B 0,C 180,E1 -19021.152,E2 -19021.152} C_VEL
LIN {X 0,Y 256.666,Z 358.597,A -85,B 0,C 180,E1 -19023.674,E2 -19023.674} C_VEL
LIN {X 0,Y 259.328,Z 350.12,A -85,B 0,C 180,E1 -19025.804,E2 -19025.804} C_VEL
LIN {X 0,Y 262.211,Z 339.922,A -85,B 0,C 180,E1 -19027.814,E2 -19027.814} C_VEL
LIN {X 0,Y 263.989,Z 332.968,A -85,B 0,C 180,E1 -19028.946,E2 -19028.946} C_VEL
LIN {X 0,Y 263.842,Z 328.555,A -85,B 0,C 180,E1 -19029.738,E2 -19029.738} C_VEL
LIN {X 0,Y 262.134,Z 317.567,A -85,B 0,C 180,E1 -19031.642,E2 -19031.642} C_VEL
LIN {X 0,Y 259.609,Z 307.378,A -85,B 0,C 180,E1 -19033.281,E2 -19033.281} C_VEL
LIN {X 0,Y 255.97,Z 296.384,A -85,B 0,C 180,E1 -19034.942,E2 -19034.942} C_VEL
LIN {X 0,Y 251.229,Z 285.246,A -85,B 0,C 180,E1 -19036.578,E2 -19036.578} C_VEL
LIN {X 0,Y 249.816,Z 282.044,A -85,B 0,C 180,E1 -19037.023,E2 -19037.023} C_VEL
LIN {X 0,Y 249.711,Z 281.351,A -85,B 0,C 180,E1 -19037.128,E2 -19037.128} C_VEL
LIN {X 0,Y 249.809,Z 279.539,A -85,B 0,C 180,E1 -19039.682,E2 -19039.682} C_VEL
LIN {X 0,Y 249.782,Z 277.993,A -85,B 0,C 180,E1 -19041.981,E2 -19041.981} C_VEL
LIN {X 0,Y 249.495,Z 275.661,A -85,B 0,C 180,E1 -19045.713,E2 -19045.713} C_VEL
LIN {X 0,Y 249.206,Z 273.485,A -85,B 0,C 180,E1 -19049.497,E2 -19049.497} C_VEL
LIN {X 0,Y 249.085,Z 272.501,A -85,B 0,C 180,E1 -19051.339,E2 -19051.339} C_VEL
LIN {X 0,Y 249.145,Z 272.448,A -85,B 0,C 180,E1 -19054.97,E2 -19054.97} C_VEL
LIN {X 0,Y 249.125,Z 272.454,A -85,B 0,C 180,E1 -19058.58,E2 -19058.58} C_VEL
LIN {X 0,Y 249.235,Z 272.44,A -85,B 0,C 180,E1 -19063.624,E2 -19063.624} C_VEL
LIN {X 0,Y 249.237,Z 272.44,A -85,B 0,C 180,E1 -19068.618,E2 -19068.618} C_VEL
LIN {X 0,Y 249.447,Z 272.412,A -85,B 0,C 180,E1 -19071.904,E2 -19071.904} C_VEL
LIN {X 0,Y 249.29,Z 272.433,A -85,B 0,C 180,E1 -19075.15,E2 -19075.15} C_VEL
LIN {X 0,Y 249.67,Z 272.386,A -85,B 0,C 180,E1 -19078.389,E2 -19078.389} C_VEL
LIN {X 0,Y 249.669,Z 272.384,A -85,B 0,C 180,E1 -19081.615,E2 -19081.615} C_VEL
LIN {X 0,Y 249.456,Z 272.412,A -85,B 0,C 180,E1 -19086.472,E2 -19086.472} C_VEL
LIN {X 0,Y 249.385,Z 272.42,A -85,B 0,C 180,E1 -19089.737,E2 -19089.737} C_VEL
LIN {X 0,Y 249.197,Z 272.447,A -85,B 0,C 180,E1 -19094.706,E2 -19094.706} C_VEL
LIN {X 0,Y 249.136,Z 272.457,A -85,B 0,C 180,E1 -19098.079,E2 -19098.079} C_VEL
LIN {X 0,Y 249.082,Z 272.465,A -85,B 0,C 180,E1 -19101.52,E2 -19101.52} C_VEL
LIN {X 0,Y 249.11,Z 272.463,A -85,B 0,C 180,E1 -19105.475,E2 -19105.475} C_VEL
LIN {X 0,Y 249.052,Z 272.467,A -85,B 0,C 180,E1 -19108.983,E2 -19108.983} C_VEL
LIN {X 0,Y 249.026,Z 272.563,A -85,B 0,C 180,E1 -19112.428,E2 -19112.428} C_VEL
LIN {X 0,Y 249.5,Z 274.922,A -85,B 0,C 180,E1 -19116.268,E2 -19116.268} C_VEL
LIN {X 0,Y 249.598,Z 275.565,A -85,B 0,C 180,E1 -19117.233,E2 -19117.233} C_VEL
LIN {X 0,Y 249.128,Z 276.613,A -85,B 0,C 180,E1 -19118.562,E2 -19118.562} C_VEL
LIN {X 0,Y 246.591,Z 278.757,A -85,B 0,C 180,E1 -19120.721,E2 -19120.721} C_VEL
LIN {X 0,Y 244.38,Z 280.561,A -85,B 0,C 180,E1 -19122.473,E2 -19122.473} C_VEL
LIN {X 0,Y 243.466,Z 281.815,A -85,B 0,C 180,E1 -19123.832,E2 -19123.832} C_VEL
LIN {X 0,Y 243.414,Z 282.193,A -85,B 0,C 180,E1 -19124.293,E2 -19124.293} C_VEL
LIN {X 0,Y 243.996,Z 285.632,A -85,B 0,C 180,E1 -19128.511,E2 -19128.511} C_VEL
LIN {X 0,Y 244.205,Z 287.817,A -85,B 0,C 180,E1 -19130.993,E2 -19130.993} C_VEL
LIN {X 0,Y 244.153,Z 290.382,A -85,B 0,C 180,E1 -19133.708,E2 -19133.708} C_VEL
LIN {X 0,Y 243.98,Z 291.608,A -85,B 0,C 180,E1 -19134.862,E2 -19134.862} C_VEL
LIN {X 0,Y 245.008,Z 294.906,A -85,B 0,C 180,E1 -19135.241,E2 -19135.241} C_VEL
LIN {X 0,Y 246.017,Z 297.253,A -85,B 0,C 180,E1 -19135.572,E2 -19135.572} C_VEL
LIN {X 0,Y 249.592,Z 307.47,A -85,B 0,C 180,E1 -19136.987,E2 -19136.987} C_VEL
LIN {X 0,Y 252.779,Z 319.816,A -85,B 0,C 180,E1 -19138.755,E2 -19138.755} C_VEL
LIN {X 0,Y 254.719,Z 331.064,A -85,B 0,C 180,E1 -19140.495,E2 -19140.495} C_VEL
LIN {X 0,Y 255.553,Z 340.743,A -85,B 0,C 180,E1 -19142.127,E2 -19142.127} C_VEL
LIN {X 0,Y 255.533,Z 350.253,A -85,B 0,C 180,E1 -19143.893,E2 -19143.893} C_VEL
LIN {X 0,Y 252.518,Z 360.206,A -85,B 0,C 180,E1 -19145.763,E2 -19145.763} C_VEL
LIN {X 0,Y 249.41,Z 369.855,A -85,B 0,C 180,E1 -19148.077,E2 -19148.077} C_VEL
LIN {X 0,Y 246.893,Z 377.599,A -85,B 0,C 180,E1 -19150.46,E2 -19150.46} C_VEL
LIN {X 0,Y 244.355,Z 384.732,A -85,B 0,C 180,E1 -19153.285,E2 -19153.285} C_VEL
LIN {X 0,Y 242.554,Z 389.524,A -85,B 0,C 180,E1 -19155.743,E2 -19155.743} C_VEL
LIN {X 0,Y 241.332,Z 393.222,A -85,B 0,C 180,E1 -19158.238,E2 -19158.238} C_VEL
LIN {X 0,Y 240.724,Z 395.146,A -85,B 0,C 180,E1 -19159.912,E2 -19159.912} C_VEL
LIN {X 0,Y 240.258,Z 396.649,A -85,B 0,C 180,E1 -19161.59,E2 -19161.59} C_VEL
LIN {X 0,Y 239.806,Z 398.403,A -85,B 0,C 180,E1 -19164.956,E2 -19164.956} C_VEL
LIN {X 0,Y 239.834,Z 398.63,A -85,B 0,C 180,E1 -19168.321,E2 -19168.321} C_VEL
LIN {X 0,Y 239.917,Z 398.118,A -85,B 0,C 180,E1 -19170,E2 -19170} C_VEL
LIN {X 0,Y 239.87,Z 397.203,A -85,B 0,C 180,E1 -19171.679,E2 -19171.679} C_VEL
LIN {X 0,Y 239.847,Z 394.275,A -85,B 0,C 180,E1 -19174.934,E2 -19174.934} C_VEL
LIN {X 0,Y 240.054,Z 390.66,A -85,B 0,C 180,E1 -19177.57,E2 -19177.57} C_VEL
LIN {X 0,Y 240.537,Z 386.058,A -85,B 0,C 180,E1 -19180.096,E2 -19180.096} C_VEL
LIN {X 0,Y 241.451,Z 379.058,A -85,B 0,C 180,E1 -19183.037,E2 -19183.037} C_VEL
LIN {X 0,Y 242.811,Z 371.481,A -85,B 0,C 180,E1 -19185.529,E2 -19185.529} C_VEL
LIN {X 0,Y 244.246,Z 362.589,A -85,B 0,C 180,E1 -19187.864,E2 -19187.864} C_VEL
LIN {X 0,Y 245.931,Z 352.063,A -85,B 0,C 180,E1 -19190.055,E2 -19190.055} C_VEL
LIN {X 0,Y 247.471,Z 342.374,A -85,B 0,C 180,E1 -19191.665,E2 -19191.665} C_VEL
LIN {X 0,Y 247.244,Z 333.252,A -85,B 0,C 180,E1 -19193.007,E2 -19193.007} C_VEL
LIN {X 0,Y 246.445,Z 322.665,A -85,B 0,C 180,E1 -19194.328,E2 -19194.328} C_VEL
LIN {X 0,Y 244.969,Z 310.662,A -85,B 0,C 180,E1 -19195.562,E2 -19195.562} C_VEL
LIN {X 0,Y 242.727,Z 298.47,A -85,B 0,C 180,E1 -19196.564,E2 -19196.564} C_VEL
LIN {X 0,Y 241.464,Z 292.38,A -85,B 0,C 180,E1 -19196.972,E2 -19196.972} C_VEL
LIN {X 0,Y 242.337,Z 287.261,A -85,B 0,C 180,E1 -19201.467,E2 -19201.467} C_VEL
LIN {X 0,Y 243.163,Z 282.967,A -85,B 0,C 180,E1 -19205.312,E2 -19205.312} C_VEL
LIN {X 0,Y 243.279,Z 280.794,A -85,B 0,C 180,E1 -19207.348,E2 -19207.348} C_VEL
LIN {X 0,Y 242.666,Z 276.978,A -85,B 0,C 180,E1 -19211.147,E2 -19211.147} C_VEL
LIN {X 0,Y 241.971,Z 273.349,A -85,B 0,C 180,E1 -19215.07,E2 -19215.07} C_VEL
LIN {X 0,Y 241.94,Z 273.352,A -85,B 0,C 180,E1 -19220.276,E2 -19220.276} C_VEL
LIN {X 0,Y 241.973,Z 273.346,A -85,B 0,C 180,E1 -19224.485,E2 -19224.485} C_VEL
LIN {X 0,Y 241.952,Z 273.348,A -85,B 0,C 180,E1 -19228.475,E2 -19228.475} C_VEL
LIN {X 0,Y 241.965,Z 273.344,A -85,B 0,C 180,E1 -19232.305,E2 -19232.305} C_VEL
LIN {X 0,Y 242.023,Z 273.335,A -85,B 0,C 180,E1 -19236.01,E2 -19236.01} C_VEL
LIN {X 0,Y 242.027,Z 273.336,A -85,B 0,C 180,E1 -19239.605,E2 -19239.605} C_VEL
LIN {X 0,Y 242.161,Z 273.317,A -85,B 0,C 180,E1 -19243.276,E2 -19243.276} C_VEL
LIN {X 0,Y 242.177,Z 273.316,A -85,B 0,C 180,E1 -19248.277,E2 -19248.277} C_VEL
LIN {X 0,Y 242.396,Z 273.291,A -85,B 0,C 180,E1 -19251.663,E2 -19251.663} C_VEL
LIN {X 0,Y 242.251,Z 273.305,A -85,B 0,C 180,E1 -19255.005,E2 -19255.005} C_VEL
LIN {X 0,Y 242.631,Z 273.243,A -85,B 0,C 180,E1 -19258.338,E2 -19258.338} C_VEL
LIN {X 0,Y 242.632,Z 273.25,A -85,B 0,C 180,E1 -19261.658,E2 -19261.658} C_VEL
LIN {X 0,Y 242.421,Z 273.286,A -85,B 0,C 180,E1 -19266.755,E2 -19266.755} C_VEL
LIN {X 0,Y 242.308,Z 273.299,A -85,B 0,C 180,E1 -19270.02,E2 -19270.02} C_VEL
LIN {X 0,Y 242.149,Z 273.321,A -85,B 0,C 180,E1 -19275.14,E2 -19275.14} C_VEL
LIN {X 0,Y 242.063,Z 273.329,A -85,B 0,C 180,E1 -19278.623,E2 -19278.623} C_VEL
LIN {X 0,Y 242.005,Z 273.336,A -85,B 0,C 180,E1 -19282.178,E2 -19282.178} C_VEL
LIN {X 0,Y 242.059,Z 273.331,A -85,B 0,C 180,E1 -19285.836,E2 -19285.836} C_VEL
LIN {X 0,Y 242.022,Z 273.332,A -85,B 0,C 180,E1 -19289.579,E2 -19289.579} C_VEL
LIN {X 0,Y 241.982,Z 273.341,A -85,B 0,C 180,E1 -19293.49,E2 -19293.49} C_VEL
LIN {X 0,Y 242.003,Z 273.336,A -85,B 0,C 180,E1 -19297.576,E2 -19297.576} C_VEL
LIN {X 0,Y 241.989,Z 273.336,A -85,B 0,C 180,E1 -19301.908,E2 -19301.908} C_VEL
LIN {X 0,Y 241.933,Z 273.346,A -85,B 0,C 180,E1 -19305.8,E2 -19305.8} C_VEL
LIN {X 0,Y 241.948,Z 273.346,A -85,B 0,C 180,E1 -19310.28,E2 -19310.28} C_VEL
LIN {X 0,Y 242.027,Z 273.338,A -85,B 0,C 180,E1 -19314.497,E2 -19314.497} C_VEL
LIN {X 0,Y 241.964,Z 273.346,A -85,B 0,C 180,E1 -19318.479,E2 -19318.479} C_VEL
LIN {X 0,Y 241.973,Z 273.345,A -85,B 0,C 180,E1 -19322.309,E2 -19322.309} C_VEL
LIN {X 0,Y 242.041,Z 273.338,A -85,B 0,C 180,E1 -19327.148,E2 -19327.148} C_VEL
LIN {X 0,Y 241.805,Z 275.193,A -85,B 0,C 180,E1 -19329.588,E2 -19329.588} C_VEL
LIN {X 0,Y 241.399,Z 279.638,A -85,B 0,C 180,E1 -19334.81,E2 -19334.81} C_VEL
LIN {X 0,Y 241.265,Z 280.951,A -85,B 0,C 180,E1 -19336.122,E2 -19336.122} C_VEL
LIN {X 0,Y 244.717,Z 293.986,A -85,B 0,C 180,E1 -19337.197,E2 -19337.197} C_VEL
LIN {X 0,Y 247.377,Z 306.887,A -85,B 0,C 180,E1 -19338.529,E2 -19338.529} C_VEL
LIN {X 0,Y 248.997,Z 319.032,A -85,B 0,C 180,E1 -19340.053,E2 -19340.053} C_VEL
LIN {X 0,Y 249.027,Z 323.487,A -85,B 0,C 180,E1 -19340.661,E2 -19340.661} C_VEL
LIN {X 0,Y 247.297,Z 334.148,A -85,B 0,C 180,E1 -19342.242,E2 -19342.242} C_VEL
LIN {X 0,Y 245.918,Z 342.867,A -85,B 0,C 180,E1 -19343.848,E2 -19343.848} C_VEL
LIN {X 0,Y 244.341,Z 351.874,A -85,B 0,C 180,E1 -19345.876,E2 -19345.876} C_VEL
LIN {X 0,Y 243.095,Z 359.302,A -85,B 0,C 180,E1 -19347.929,E2 -19347.929} C_VEL
LIN {X 0,Y 241.765,Z 366.626,A -85,B 0,C 180,E1 -19350.416,E2 -19350.416} C_VEL
LIN {X 0,Y 241.065,Z 371.569,A -85,B 0,C 180,E1 -19352.506,E2 -19352.506} C_VEL
LIN {X 0,Y 240.468,Z 376.377,A -85,B 0,C 180,E1 -19355.03,E2 -19355.03} C_VEL
LIN {X 0,Y 239.976,Z 380.081,A -85,B 0,C 180,E1 -19357.573,E2 -19357.573} C_VEL
LIN {X 0,Y 239.642,Z 382.764,A -85,B 0,C 180,E1 -19360.134,E2 -19360.134} C_VEL
LIN {X 0,Y 239.556,Z 384.03,A -85,B 0,C 180,E1 -19361.85,E2 -19361.85} C_VEL
LIN {X 0,Y 239.658,Z 385.165,A -85,B 0,C 180,E1 -19364.605,E2 -19364.605} C_VEL
LIN {X 0,Y 239.797,Z 385.275,A -85,B 0,C 180,E1 -19367.042,E2 -19367.042} C_VEL
LIN {X 0,Y 240.146,Z 384.881,A -85,B 0,C 180,E1 -19368.779,E2 -19368.779} C_VEL
LIN {X 0,Y 240.726,Z 383.776,A -85,B 0,C 180,E1 -19370.901,E2 -19370.901} C_VEL
LIN {X 0,Y 241.894,Z 381.044,A -85,B 0,C 180,E1 -19374.001,E2 -19374.001} C_VEL
LIN {X 0,Y 243.195,Z 377.878,A -85,B 0,C 180,E1 -19376.387,E2 -19376.387} C_VEL
LIN {X 0,Y 245.146,Z 372.928,A -85,B 0,C 180,E1 -19379.167,E2 -19379.167} C_VEL
LIN {X 0,Y 247.527,Z 366.439,A -85,B 0,C 180,E1 -19381.892,E2 -19381.892} C_VEL
LIN {X 0,Y 250.033,Z 359.386,A -85,B 0,C 180,E1 -19384.205,E2 -19384.205} C_VEL
LIN {X 0,Y 252.889,Z 350.756,A -85,B 0,C 180,E1 -19386.452,E2 -19386.452} C_VEL
LIN {X 0,Y 255.772,Z 341.065,A -85,B 0,C 180,E1 -19388.438,E2 -19388.438} C_VEL
LIN {X 0,Y 257.676,Z 334.012,A -85,B 0,C 180,E1 -19389.624,E2 -19389.624} C_VEL
LIN {X 0,Y 256.966,Z 326.052,A -85,B 0,C 180,E1 -19391.141,E2 -19391.141} C_VEL
LIN {X 0,Y 255.188,Z 315.995,A -85,B 0,C 180,E1 -19392.929,E2 -19392.929} C_VEL
LIN {X 0,Y 252.263,Z 305.232,A -85,B 0,C 180,E1 -19394.734,E2 -19394.734} C_VEL
LIN {X 0,Y 247.97,Z 293.35,A -85,B 0,C 180,E1 -19396.633,E2 -19396.633} C_VEL
LIN {X 0,Y 244.314,Z 285.439,A -85,B 0,C 180,E1 -19397.889,E2 -19397.889} C_VEL
LIN {X 0,Y 242.943,Z 282.532,A -85,B 0,C 180,E1 -19398.338,E2 -19398.338} C_VEL
LIN {X 0,Y 242.743,Z 281.648,A -85,B 0,C 180,E1 -19398.432,E2 -19398.432} C_VEL
LIN {X 0,Y 242.795,Z 279.655,A -85,B 0,C 180,E1 -19401.401,E2 -19401.401} C_VEL
LIN {X 0,Y 242.61,Z 277.667,A -85,B 0,C 180,E1 -19404.597,E2 -19404.597} C_VEL
LIN {X 0,Y 242.305,Z 275.413,A -85,B 0,C 180,E1 -19408.53,E2 -19408.53} C_VEL
LIN {X 0,Y 242.029,Z 273.46,A -85,B 0,C 180,E1 -19412.318,E2 -19412.318} C_VEL
LIN {X 0,Y 242.061,Z 273.335,A -85,B 0,C 180,E1 -19416.019,E2 -19416.019} C_VEL
LIN {X 0,Y 242.065,Z 273.328,A -85,B 0,C 180,E1 -19419.613,E2 -19419.613} C_VEL
LIN {X 0,Y 242.156,Z 273.319,A -85,B 0,C 180,E1 -19423.28,E2 -19423.28} C_VEL
LIN {X 0,Y 242.173,Z 273.319,A -85,B 0,C 180,E1 -19428.281,E2 -19428.281} C_VEL
LIN {X 0,Y 242.393,Z 273.291,A -85,B 0,C 180,E1 -19431.666,E2 -19431.666} C_VEL
LIN {X 0,Y 242.251,Z 273.31,A -85,B 0,C 180,E1 -19435.009,E2 -19435.009} C_VEL
LIN {X 0,Y 242.63,Z 273.263,A -85,B 0,C 180,E1 -19438.342,E2 -19438.342} C_VEL
LIN {X 0,Y 242.63,Z 273.261,A -85,B 0,C 180,E1 -19441.662,E2 -19441.662} C_VEL
LIN {X 0,Y 242.428,Z 273.289,A -85,B 0,C 180,E1 -19446.661,E2 -19446.661} C_VEL
LIN {X 0,Y 242.31,Z 273.301,A -85,B 0,C 180,E1 -19450.024,E2 -19450.024} C_VEL
LIN {X 0,Y 242.161,Z 273.323,A -85,B 0,C 180,E1 -19455.143,E2 -19455.143} C_VEL
LIN {X 0,Y 242.07,Z 273.337,A -85,B 0,C 180,E1 -19458.626,E2 -19458.626} C_VEL
LIN {X 0,Y 242.004,Z 273.347,A -85,B 0,C 180,E1 -19462.183,E2 -19462.183} C_VEL
LIN {X 0,Y 242.048,Z 273.341,A -85,B 0,C 180,E1 -19465.832,E2 -19465.832} C_VEL
LIN {X 0,Y 241.974,Z 273.348,A -85,B 0,C 180,E1 -19469.59,E2 -19469.59} C_VEL
LIN {X 0,Y 242.014,Z 273.658,A -85,B 0,C 180,E1 -19471.516,E2 -19471.516} C_VEL
LIN {X 0,Y 242.51,Z 276.141,A -85,B 0,C 180,E1 -19475.764,E2 -19475.764} C_VEL
LIN {X 0,Y 242.897,Z 278.648,A -85,B 0,C 180,E1 -19479.537,E2 -19479.537} C_VEL
LIN {X 0,Y 243.174,Z 280.186,A -85,B 0,C 180,E1 -19481.664,E2 -19481.664} C_VEL
LIN {X 0,Y 243.414,Z 282.193,A -85,B 0,C 180,E1 -19484.293,E2 -19484.293} C_VEL
LIN {X 0,Y 242.865,Z 283.405,A -85,B 0,C 180,E1 -19485.649,E2 -19485.649} C_VEL
LIN {X 0,Y 240.289,Z 285.743,A -85,B 0,C 180,E1 -19487.852,E2 -19487.852} C_VEL
LIN {X 0,Y 238.108,Z 287.685,A -85,B 0,C 180,E1 -19489.642,E2 -19489.642} C_VEL
LIN {X 0,Y 237.233,Z 289.06,A -85,B 0,C 180,E1 -19491.029,E2 -19491.029} C_VEL
LIN {X 0,Y 237.196,Z 289.485,A -85,B 0,C 180,E1 -19491.499,E2 -19491.499} C_VEL
LIN {X 0,Y 237.154,Z 291.238,A -85,B 0,C 180,E1 -19493.419,E2 -19493.419} C_VEL
LIN {X 0,Y 238.294,Z 294.793,A -85,B 0,C 180,E1 -19493.886,E2 -19493.886} C_VEL
LIN {X 0,Y 239.254,Z 296.879,A -85,B 0,C 180,E1 -19494.214,E2 -19494.214} C_VEL
LIN {X 0,Y 243.323,Z 308.138,A -85,B 0,C 180,E1 -19495.897,E2 -19495.897} C_VEL
LIN {X 0,Y 246.354,Z 319.948,A -85,B 0,C 180,E1 -19497.689,E2 -19497.689} C_VEL
LIN {X 0,Y 248.373,Z 332.082,A -85,B 0,C 180,E1 -19499.677,E2 -19499.677} C_VEL
LIN {X 0,Y 249.131,Z 341.472,A -85,B 0,C 180,E1 -19501.343,E2 -19501.343} C_VEL
LIN {X 0,Y 249.082,Z 350.808,A -85,B 0,C 180,E1 -19503.164,E2 -19503.164} C_VEL
LIN {X 0,Y 246.716,Z 358.844,A -85,B 0,C 180,E1 -19504.705,E2 -19504.705} C_VEL
LIN {X 0,Y 243.848,Z 367.215,A -85,B 0,C 180,E1 -19506.654,E2 -19506.654} C_VEL
LIN {X 0,Y 240.872,Z 375.818,A -85,B 0,C 180,E1 -19509.209,E2 -19509.209} C_VEL
LIN {X 0,Y 238.332,Z 383.027,A -85,B 0,C 180,E1 -19511.964,E2 -19511.964} C_VEL
LIN {X 0,Y 236.231,Z 388.136,A -85,B 0,C 180,E1 -19514.47,E2 -19514.47} C_VEL
LIN {X 0,Y 234.765,Z 392.124,A -85,B 0,C 180,E1 -19517.026,E2 -19517.026} C_VEL
LIN {X 0,Y 233.722,Z 395.093,A -85,B 0,C 180,E1 -19519.606,E2 -19519.606} C_VEL
LIN {X 0,Y 233.225,Z 396.543,A -85,B 0,C 180,E1 -19521.335,E2 -19521.335} C_VEL
LIN {X 0,Y 232.737,Z 398.243,A -85,B 0,C 180,E1 -19524.803,E2 -19524.803} C_VEL
LIN {X 0,Y 232.675,Z 398.522,A -85,B 0,C 180,E1 -19526.537,E2 -19526.537} C_VEL
LIN {X 0,Y 232.746,Z 398.397,A -85,B 0,C 180,E1 -19528.27,E2 -19528.27} C_VEL
LIN {X 0,Y 232.848,Z 397.852,A -85,B 0,C 180,E1 -19530,E2 -19530} C_VEL
LIN {X 0,Y 232.781,Z 396.909,A -85,B 0,C 180,E1 -19531.73,E2 -19531.73} C_VEL
LIN {X 0,Y 232.763,Z 394.173,A -85,B 0,C 180,E1 -19534.847,E2 -19534.847} C_VEL
LIN {X 0,Y 233.007,Z 390.232,A -85,B 0,C 180,E1 -19537.801,E2 -19537.801} C_VEL
LIN {X 0,Y 233.518,Z 385.559,A -85,B 0,C 180,E1 -19540.403,E2 -19540.403} C_VEL
LIN {X 0,Y 234.507,Z 378.484,A -85,B 0,C 180,E1 -19543.43,E2 -19543.43} C_VEL
LIN {X 0,Y 235.919,Z 370.822,A -85,B 0,C 180,E1 -19545.995,E2 -19545.995} C_VEL
LIN {X 0,Y 237.283,Z 362.506,A -85,B 0,C 180,E1 -19548.228,E2 -19548.228} C_VEL
LIN {X 0,Y 239.03,Z 352.224,A -85,B 0,C 180,E1 -19550.435,E2 -19550.435} C_VEL
LIN {X 0,Y 240.63,Z 342.612,A -85,B 0,C 180,E1 -19552.088,E2 -19552.088} C_VEL
LIN {X 0,Y 240.291,Z 331.911,A -85,B 0,C 180,E1 -19553.713,E2 -19553.713} C_VEL
LIN {X 0,Y 239.303,Z 319.935,A -85,B 0,C 180,E1 -19555.204,E2 -19555.204} C_VEL
LIN {X 0,Y 237.487,Z 306.763,A -85,B 0,C 180,E1 -19556.523,E2 -19556.523} C_VEL
LIN {X 0,Y 234.73,Z 293.72,A -85,B 0,C 180,E1 -19557.57,E2 -19557.57} C_VEL
LIN {X 0,Y 234.497,Z 292.154,A -85,B 0,C 180,E1 -19557.683,E2 -19557.683} C_VEL
LIN {X 0,Y 235.483,Z 286.873,A -85,B 0,C 180,E1 -19562.493,E2 -19562.493} C_VEL
LIN {X 0,Y 236.131,Z 283.654,A -85,B 0,C 180,E1 -19565.476,E2 -19565.476} C_VEL
LIN {X 0,Y 236.221,Z 281.464,A -85,B 0,C 180,E1 -19567.581,E2 -19567.581} C_VEL
LIN {X 0,Y 235.565,Z 277.426,A -85,B 0,C 180,E1 -19571.764,E2 -19571.764} C_VEL
LIN {X 0,Y 234.91,Z 274.229,A -85,B 0,C 180,E1 -19575.326,E2 -19575.326} C_VEL
LIN {X 0,Y 234.854,Z 274.237,A -85,B 0,C 180,E1 -19578.824,E2 -19578.824} C_VEL
LIN {X 0,Y 234.919,Z 274.227,A -85,B 0,C 180,E1 -19581.077,E2 -19581.077} C_VEL
LIN {X 0,Y 234.922,Z 274.221,A -85,B 0,C 180,E1 -19585.359,E2 -19585.359} C_VEL
LIN {X 0,Y 234.898,Z 274.221,A -85,B 0,C 180,E1 -19589.425,E2 -19589.425} C_VEL
LIN {X 0,Y 234.968,Z 274.215,A -85,B 0,C 180,E1 -19593.805,E2 -19593.805} C_VEL
LIN {X 0,Y 234.991,Z 274.213,A -85,B 0,C 180,E1 -19598.966,E2 -19598.966} C_VEL
LIN {X 0,Y 235.094,Z 274.198,A -85,B 0,C 180,E1 -19603.058,E2 -19603.058} C_VEL
LIN {X 0,Y 235.11,Z 274.198,A -85,B 0,C 180,E1 -19607.92,E2 -19607.92} C_VEL
LIN {X 0,Y 235.328,Z 274.171,A -85,B 0,C 180,E1 -19611.41,E2 -19611.41} C_VEL
LIN {X 0,Y 235.369,Z 274.166,A -85,B 0,C 180,E1 -19613.138,E2 -19613.138} C_VEL
LIN {X 0,Y 235.591,Z 274.119,A -85,B 0,C 180,E1 -19618.289,E2 -19618.289} C_VEL
LIN {X 0,Y 235.591,Z 274.127,A -85,B 0,C 180,E1 -19621.707,E2 -19621.707} C_VEL
LIN {X 0,Y 235.398,Z 274.161,A -85,B 0,C 180,E1 -19626.857,E2 -19626.857} C_VEL
LIN {X 0,Y 235.232,Z 274.179,A -85,B 0,C 180,E1 -19630.325,E2 -19630.325} C_VEL
LIN {X 0,Y 235.1,Z 274.197,A -85,B 0,C 180,E1 -19635.605,E2 -19635.605} C_VEL
LIN {X 0,Y 235,Z 274.211,A -85,B 0,C 180,E1 -19639.204,E2 -19639.204} C_VEL
LIN {X 0,Y 234.954,Z 274.215,A -85,B 0,C 180,E1 -19642.881,E2 -19642.881} C_VEL
LIN {X 0,Y 234.962,Z 274.215,A -85,B 0,C 180,E1 -19646.656,E2 -19646.656} C_VEL
LIN {X 0,Y 234.924,Z 274.215,A -85,B 0,C 180,E1 -19650.566,E2 -19650.566} C_VEL
LIN {X 0,Y 234.952,Z 274.216,A -85,B 0,C 180,E1 -19654.631,E2 -19654.631} C_VEL
LIN {X 0,Y 234.958,Z 274.217,A -85,B 0,C 180,E1 -19658.951,E2 -19658.951} C_VEL
LIN {X 0,Y 234.965,Z 274.214,A -85,B 0,C 180,E1 -19663.465,E2 -19663.465} C_VEL
LIN {X 0,Y 234.878,Z 274.223,A -85,B 0,C 180,E1 -19668.418,E2 -19668.418} C_VEL
LIN {X 0,Y 234.912,Z 274.222,A -85,B 0,C 180,E1 -19671.078,E2 -19671.078} C_VEL
LIN {X 0,Y 234.951,Z 274.217,A -85,B 0,C 180,E1 -19675.366,E2 -19675.366} C_VEL
LIN {X 0,Y 234.911,Z 274.222,A -85,B 0,C 180,E1 -19679.43,E2 -19679.43} C_VEL
LIN {X 0,Y 234.934,Z 274.22,A -85,B 0,C 180,E1 -19683.818,E2 -19683.818} C_VEL
LIN {X 0,Y 235.018,Z 274.363,A -85,B 0,C 180,E1 -19687.395,E2 -19687.395} C_VEL
LIN {X 0,Y 234.443,Z 278.552,A -85,B 0,C 180,E1 -19692.556,E2 -19692.556} C_VEL
LIN {X 0,Y 234.289,Z 280.983,A -85,B 0,C 180,E1 -19695.422,E2 -19695.422} C_VEL
LIN {X 0,Y 237.718,Z 294.088,A -85,B 0,C 180,E1 -19696.541,E2 -19696.541} C_VEL
LIN {X 0,Y 240.393,Z 306.54,A -85,B 0,C 180,E1 -19697.878,E2 -19697.878} C_VEL
LIN {X 0,Y 241.952,Z 317.928,A -85,B 0,C 180,E1 -19699.329,E2 -19699.329} C_VEL
LIN {X 0,Y 242.38,Z 322.419,A -85,B 0,C 180,E1 -19699.981,E2 -19699.981} C_VEL
LIN {X 0,Y 240.641,Z 333.374,A -85,B 0,C 180,E1 -19701.603,E2 -19701.603} C_VEL
LIN {X 0,Y 238.901,Z 344.199,A -85,B 0,C 180,E1 -19703.666,E2 -19703.666} C_VEL
LIN {X 0,Y 237.246,Z 353.027,A -85,B 0,C 180,E1 -19705.753,E2 -19705.753} C_VEL
LIN {X 0,Y 235.974,Z 360.296,A -85,B 0,C 180,E1 -19707.866,E2 -19707.866} C_VEL
LIN {X 0,Y 234.664,Z 367.468,A -85,B 0,C 180,E1 -19710.429,E2 -19710.429} C_VEL
LIN {X 0,Y 233.932,Z 372.301,A -85,B 0,C 180,E1 -19712.583,E2 -19712.583} C_VEL
LIN {X 0,Y 233.332,Z 376.998,A -85,B 0,C 180,E1 -19715.184,E2 -19715.184} C_VEL
LIN {X 0,Y 232.825,Z 380.6,A -85,B 0,C 180,E1 -19717.807,E2 -19717.807} C_VEL
